C01799=1037.388,344.566,-126.186,172.352,44.021,158.561
C01800=1037.395,344.814,-126.222,172.357,44.023,158.563
C01801=1037.403,345.061,-126.259,172.364,44.026,158.564
C01802=1037.410,345.308,-126.297,172.369,44.028,158.565
C01803=1037.418,345.555,-126.334,172.375,44.031,158.566
C01804=1037.425,345.802,-126.371,172.380,44.033,158.567
C01805=1037.433,346.049,-126.408,172.385,44.036,158.568
C01806=1037.440,346.296,-126.445,172.391,44.039,158.569
C01807=1037.447,346.544,-126.483,172.396,44.041,158.570
C01808=1037.455,346.790,-126.520,172.402,44.043,158.571
C01809=1037.463,347.038,-126.557,172.408,44.046,158.573
C01810=1037.470,347.284,-126.594,172.413,44.049,158.574
C01811=1037.478,347.531,-126.632,172.419,44.051,158.575
C01812=1037.486,347.779,-126.669,172.424,44.054,158.576
C01813=1037.494,348.026,-126.706,172.431,44.057,158.577
C01814=1037.501,348.273,-126.744,172.436,44.059,158.578
C01815=1037.513,348.639,-126.800,172.444,44.063,158.580
C01816=1037.524,349.005,-126.855,172.452,44.067,158.581
C01817=1037.535,349.371,-126.911,172.461,44.071,158.583
C01818=1037.546,349.738,-126.966,172.470,44.075,158.585
C01819=1037.554,349.984,-127.004,172.475,44.077,158.586
C01820=1037.561,350.231,-127.042,172.480,44.080,158.587
C01821=1037.569,350.478,-127.079,172.487,44.083,158.588
C01822=1037.577,350.725,-127.117,172.492,44.085,158.589
C01823=1037.584,350.973,-127.155,172.498,44.089,158.591
C01824=1037.592,351.220,-127.192,172.503,44.092,158.592
C01825=1037.599,351.466,-127.231,172.510,44.094,158.593
C01826=1037.607,351.714,-127.269,172.515,44.097,158.594
C01827=1037.615,351.960,-127.306,172.521,44.100,158.595
C01828=1037.623,352.207,-127.344,172.526,44.102,158.596
C01829=1037.631,352.455,-127.382,172.533,44.105,158.598
C01830=1037.638,352.702,-127.420,172.538,44.108,158.599
C01831=1037.645,352.948,-127.458,172.544,44.111,158.600
C01832=1037.653,353.196,-127.496,172.550,44.114,158.601
C01833=1037.661,353.443,-127.534,172.556,44.116,158.602
C01834=1037.668,353.689,-127.573,172.561,44.119,158.604
C01835=1037.677,353.937,-127.610,172.568,44.122,158.605
C01836=1037.685,354.183,-127.648,172.574,44.125,158.606
C01837=1037.692,354.431,-127.686,172.579,44.128,158.607
C01838=1037.700,354.678,-127.724,172.586,44.130,158.608
C01839=1037.708,354.924,-127.762,172.591,44.134,158.610
C01840=1037.716,355.171,-127.801,172.598,44.136,158.611
C01841=1037.723,355.418,-127.839,172.603,44.139,158.612
C01842=1037.731,355.666,-127.877,172.609,44.142,158.613
C01843=1037.739,355.912,-127.915,172.616,44.145,158.615
C01844=1037.747,356.159,-127.953,172.621,44.148,158.616
C01845=1037.754,356.406,-127.992,172.628,44.151,158.617
C01846=1037.762,356.653,-128.031,172.633,44.154,158.619
C01847=1037.770,356.900,-128.069,172.639,44.157,158.620
C01848=1037.778,357.147,-128.108,172.646,44.160,158.621
C01849=1037.786,357.393,-128.146,172.651,44.163,158.622
C01850=1037.794,357.641,-128.185,172.658,44.166,158.624
C01851=1037.801,357.887,-128.223,172.663,44.168,158.625
C01852=1037.810,358.134,-128.261,172.670,44.172,158.626
C01853=1037.818,358.381,-128.300,172.676,44.175,158.627
C01854=1037.825,358.628,-128.338,172.681,44.178,158.629
C01855=1037.833,358.875,-128.377,172.688,44.181,158.630
C01856=1037.841,359.122,-128.415,172.694,44.184,158.631
C01857=1037.848,359.369,-128.454,172.700,44.187,158.632
C01858=1037.857,359.616,-128.494,172.706,44.190,158.634
C01859=1037.864,359.862,-128.532,172.713,44.193,158.635
C01860=1037.873,360.110,-128.571,172.718,44.196,158.636
C01861=1037.881,360.356,-128.610,172.725,44.199,158.638
C01862=1037.889,360.603,-128.648,172.731,44.202,158.639
C01863=1037.897,360.850,-128.687,172.737,44.205,158.640
C01864=1037.904,361.097,-128.727,172.744,44.208,158.642
C01865=1037.912,361.343,-128.765,172.750,44.212,158.643
C01866=1037.920,361.591,-128.804,172.757,44.215,158.644
C01867=1037.929,361.837,-128.843,172.762,44.218,158.646
C01868=1037.937,362.084,-128.881,172.769,44.221,158.647
C01869=1037.944,362.331,-128.921,172.775,44.225,158.648
C01870=1037.952,362.578,-128.960,172.782,44.228,158.650
C01871=1037.964,362.950,-129.019,172.791,44.233,158.652
C01872=1037.975,363.322,-129.078,172.801,44.237,158.654
C01873=1037.988,363.694,-129.138,172.811,44.242,158.656
C01874=1037.999,364.067,-129.197,172.819,44.248,158.658
C01875=1038.008,364.313,-129.236,172.826,44.251,158.659
C01876=1038.016,364.560,-129.276,172.833,44.254,158.661
C01877=1038.023,364.806,-129.315,172.839,44.258,158.662
C01878=1038.031,365.053,-129.355,172.846,44.261,158.664
C01879=1038.039,365.300,-129.393,172.852,44.264,158.665
C01880=1038.048,365.547,-129.433,172.858,44.267,158.666
C01881=1038.056,365.794,-129.473,172.865,44.271,158.668
C01882=1038.064,366.040,-129.512,172.872,44.274,158.669
C01883=1038.072,366.287,-129.552,172.877,44.277,158.671
C01884=1038.080,366.534,-129.591,172.884,44.281,158.672
C01885=1038.088,366.781,-129.631,172.891,44.284,158.674
C01886=1038.096,367.027,-129.670,172.897,44.288,158.675
C01887=1038.104,367.274,-129.710,172.904,44.291,158.676
C01888=1038.113,367.521,-129.750,172.911,44.295,158.678
C01889=1038.121,367.767,-129.789,172.917,44.298,158.679
C01890=1038.129,368.014,-129.829,172.924,44.302,158.681
C01891=1038.137,368.260,-129.869,172.931,44.305,158.682
C01892=1038.145,368.507,-129.909,172.938,44.308,158.684
C01893=1038.154,368.754,-129.948,172.943,44.312,158.685
C01894=1038.161,369.001,-129.988,172.950,44.315,158.687
C01895=1038.170,369.247,-130.027,172.957,44.318,158.688
C01896=1038.178,369.493,-130.068,172.964,44.322,158.690
C01897=1038.186,369.740,-130.107,172.971,44.326,158.691
C01898=1038.195,369.988,-130.148,172.977,44.329,158.692
C01899=1038.203,370.234,-130.188,172.984,44.333,158.694
C01900=1038.211,370.480,-130.228,172.991,44.336,158.696
C01901=1038.219,370.727,-130.268,172.998,44.340,158.697
C01902=1038.228,370.973,-130.308,173.005,44.343,158.699
C01903=1038.236,371.220,-130.348,173.011,44.347,158.700
C01904=1038.243,371.467,-130.388,173.018,44.351,158.702
C01905=1038.251,371.713,-130.429,173.025,44.355,158.703
C01906=1038.260,371.960,-130.470,173.032,44.358,158.705
C01907=1038.268,372.206,-130.509,173.039,44.362,158.706
C01908=1038.276,372.453,-130.550,173.046,44.366,158.708
C01909=1038.285,372.699,-130.590,173.053,44.369,158.709
C01910=1038.293,372.947,-130.631,173.059,44.373,158.711
C01911=1038.302,373.193,-130.671,173.066,44.377,158.712
C01912=1038.310,373.439,-130.711,173.073,44.380,158.714
C01913=1038.318,373.685,-130.752,173.080,44.384,158.716
C01914=1038.326,373.932,-130.793,173.087,44.388,158.717
C01915=1038.334,374.179,-130.833,173.094,44.391,158.719
C01916=1038.343,374.425,-130.873,173.101,44.395,158.720
C01917=1038.351,374.672,-130.914,173.108,44.399,158.722
C01918=1038.359,374.918,-130.955,173.115,44.403,158.724
C01919=1038.367,375.165,-130.995,173.122,44.406,158.725
C01920=1038.376,375.412,-131.036,173.130,44.411,158.727
C01921=1038.384,375.658,-131.077,173.137,44.414,158.728
C01922=1038.393,375.904,-131.117,173.144,44.418,158.730
C01923=1038.401,376.151,-131.158,173.151,44.422,158.732
C01924=1038.410,376.397,-131.199,173.158,44.426,158.733
C01925=1038.418,376.643,-131.240,173.165,44.429,158.735
C01926=1038.426,376.890,-131.281,173.172,44.433,158.736
C01927=1038.441,377.283,-131.346,173.184,44.439,158.739
C01928=1038.454,377.675,-131.410,173.195,44.446,158.742
C01929=1038.468,378.068,-131.476,173.207,44.452,158.744
C01930=1038.482,378.461,-131.541,173.218,44.458,158.747
C01931=1038.489,378.707,-131.583,173.225,44.462,158.749
C01932=1038.498,378.954,-131.624,173.233,44.467,158.750
C01933=1038.506,379.200,-131.665,173.240,44.470,158.752
C01934=1038.515,379.447,-131.706,173.247,44.474,158.754
C01935=1038.523,379.692,-131.748,173.254,44.478,158.755
C01936=1038.532,379.939,-131.789,173.261,44.483,158.757
C01937=1038.541,380.184,-131.831,173.270,44.487,158.759
C01938=1038.549,380.431,-131.872,173.277,44.491,158.761
C01939=1038.558,380.677,-131.913,173.284,44.495,158.762
C01940=1038.566,380.923,-131.955,173.292,44.499,158.764
C01941=1038.574,381.169,-131.997,173.299,44.503,158.766
C01942=1038.583,381.416,-132.038,173.306,44.507,158.768
C01943=1038.591,381.662,-132.079,173.315,44.511,158.769
C01944=1038.600,381.908,-132.121,173.322,44.516,158.771
C01945=1038.609,382.155,-132.162,173.329,44.520,158.773
C01946=1038.618,382.401,-132.204,173.336,44.524,158.775
C01947=1038.625,382.647,-132.246,173.344,44.528,158.776
C01948=1038.634,382.893,-132.288,173.352,44.532,158.778
C01949=1038.643,383.140,-132.330,173.360,44.537,158.780
C01950=1038.652,383.386,-132.371,173.367,44.541,158.782
C01951=1038.661,383.633,-132.413,173.374,44.545,158.783
C01952=1038.669,383.878,-132.454,173.383,44.549,158.785
C01953=1038.678,384.125,-132.497,173.390,44.554,158.787
C01954=1038.687,384.371,-132.538,173.397,44.558,158.789
C01955=1038.696,384.618,-132.580,173.406,44.562,158.791
C01956=1038.704,384.864,-132.622,173.413,44.567,158.793
C01957=1038.714,385.110,-132.664,173.421,44.571,158.794
C01958=1038.722,385.356,-132.707,173.428,44.575,158.796
C01959=1038.731,385.603,-132.748,173.436,44.579,158.798
C01960=1038.740,385.849,-132.790,173.444,44.584,158.800
C01961=1038.749,386.095,-132.832,173.452,44.588,158.802
C01962=1038.758,386.341,-132.874,173.460,44.593,158.804
C01963=1038.766,386.588,-132.916,173.467,44.597,158.805
C01964=1038.775,386.834,-132.959,173.476,44.601,158.807
C01965=1038.784,387.080,-133.001,173.483,44.606,158.809
C01966=1038.794,387.326,-133.043,173.492,44.610,158.811
C01967=1038.802,387.572,-133.085,173.499,44.615,158.813
C01968=1038.811,387.818,-133.128,173.508,44.619,158.815
C01969=1038.820,388.065,-133.169,173.515,44.624,158.817
C01970=1038.829,388.311,-133.213,173.523,44.628,158.819
C01971=1038.838,388.557,-133.255,173.531,44.632,158.821
C01972=1038.847,388.803,-133.297,173.539,44.637,158.823
C01973=1038.856,389.050,-133.340,173.548,44.642,158.825
C01974=1038.865,389.295,-133.382,173.555,44.646,158.826
C01975=1038.873,389.541,-133.426,173.564,44.651,158.828
C01976=1038.883,389.787,-133.468,173.571,44.655,158.830
C01977=1038.892,390.034,-133.511,173.580,44.660,158.832
C01978=1038.901,390.280,-133.553,173.588,44.665,158.834
C01979=1038.909,390.526,-133.596,173.596,44.670,158.836
C01980=1038.918,390.772,-133.639,173.604,44.674,158.838
C01981=1038.928,391.019,-133.682,173.613,44.679,158.840
C01982=1038.937,391.264,-133.724,173.621,44.684,158.842
C01983=1038.945,391.477,-133.762,173.627,44.687,158.844
C01984=1038.952,391.691,-133.799,173.635,44.692,158.846
C01985=1038.959,391.904,-133.837,173.642,44.696,158.847
C01986=1038.967,392.117,-133.874,173.649,44.700,158.849
C01987=1038.976,392.331,-133.912,173.657,44.704,158.851
C01988=1038.983,392.544,-133.949,173.664,44.709,158.853
C01989=1038.991,392.757,-133.986,173.672,44.713,158.855
C01990=1038.999,392.971,-134.024,173.679,44.717,158.856
C01991=1039.009,393.217,-134.067,173.687,44.721,158.858
C01992=1039.017,393.463,-134.110,173.696,44.726,158.861
C01993=1039.026,393.709,-134.154,173.704,44.731,158.863
C01994=1039.036,393.955,-134.196,173.712,44.736,158.865
C01995=1039.045,394.201,-134.240,173.721,44.741,158.867
C01996=1039.054,394.447,-134.283,173.730,44.746,158.869
C01997=1039.064,394.693,-134.327,173.737,44.751,158.871
C01998=1039.072,394.939,-134.370,173.746,44.756,158.873
C01999=1039.082,395.185,-134.414,173.755,44.761,158.875
C02000=1039.091,395.430,-134.457,173.764,44.766,158.877
C02001=1039.100,395.677,-134.501,173.772,44.771,158.879
C02002=1039.109,395.922,-134.544,173.781,44.776,158.882
C02003=1039.119,396.168,-134.588,173.790,44.781,158.884
C02004=1039.127,396.414,-134.632,173.799,44.786,158.886
C02005=1039.136,396.660,-134.676,173.807,44.791,158.888
C02006=1039.147,396.906,-134.719,173.815,44.796,158.890
C02007=1039.155,397.152,-134.763,173.824,44.801,158.892
C02008=1039.165,397.398,-134.807,173.833,44.806,158.895
C02009=1039.174,397.644,-134.851,173.842,44.811,158.897
C02010=1039.183,397.889,-134.895,173.851,44.816,158.899
C02011=1039.192,398.136,-134.939,173.860,44.821,158.901
C02012=1039.203,398.381,-134.982,173.869,44.826,158.903
C02013=1039.212,398.627,-135.027,173.878,44.832,158.906
C02014=1039.221,398.873,-135.070,173.887,44.837,158.908
C02015=1039.231,399.118,-135.115,173.896,44.842,158.910
C02016=1039.240,399.365,-135.159,173.904,44.848,158.912
C02017=1039.249,399.611,-135.203,173.913,44.853,158.914
C02018=1039.259,399.857,-135.247,173.922,44.858,158.917
C02019=1039.268,400.102,-135.292,173.931,44.863,158.919
C02020=1039.277,400.348,-135.336,173.940,44.868,158.921
C02021=1039.287,400.594,-135.380,173.949,44.874,158.924
C02022=1039.296,400.839,-135.425,173.958,44.879,158.926
C02023=1039.306,401.086,-135.469,173.968,44.884,158.928
C02024=1039.316,401.331,-135.514,173.978,44.890,158.931
C02025=1039.325,401.577,-135.558,173.987,44.895,158.933
C02026=1039.335,401.823,-135.603,173.996,44.901,158.935
C02027=1039.344,402.068,-135.648,174.005,44.906,158.938
C02028=1039.354,402.314,-135.692,174.014,44.911,158.940
C02029=1039.363,402.560,-135.737,174.023,44.917,158.942
C02030=1039.373,402.805,-135.781,174.032,44.922,158.945
C02031=1039.382,403.051,-135.827,174.042,44.928,158.947
C02032=1039.392,403.298,-135.871,174.051,44.934,158.949
C02033=1039.402,403.544,-135.916,174.061,44.939,158.952
C02034=1039.412,403.789,-135.961,174.070,44.944,158.954
C02035=1039.421,404.035,-136.006,174.080,44.950,158.957
C02036=1039.430,404.280,-136.051,174.089,44.956,158.959
C02037=1039.440,404.526,-136.096,174.098,44.961,158.961
C02038=1039.450,404.771,-136.141,174.108,44.967,158.964
C02039=1039.459,405.018,-136.187,174.118,44.973,158.966
C02040=1039.469,405.263,-136.232,174.127,44.978,158.969
C02041=1039.479,405.508,-136.277,174.137,44.984,158.971
C02042=1039.488,405.754,-136.322,174.147,44.989,158.974
C02043=1039.498,405.978,-136.363,174.155,44.995,158.976
C02044=1039.506,406.201,-136.405,174.164,45.000,158.978
C02045=1039.515,406.424,-136.446,174.173,45.005,158.981
C02046=1039.525,406.647,-136.487,174.182,45.010,158.983
C02047=1039.533,406.870,-136.529,174.190,45.016,158.985
C02048=1039.542,407.093,-136.569,174.199,45.021,158.987
C02049=1039.551,407.317,-136.611,174.208,45.026,158.990
C02050=1039.560,407.540,-136.653,174.218,45.032,158.992
C02051=1039.570,407.786,-136.698,174.227,45.038,158.995
C02052=1039.580,408.031,-136.744,174.238,45.043,158.997
C02053=1039.590,408.277,-136.789,174.247,45.049,159.000
C02054=1039.599,408.523,-136.835,174.257,45.055,159.002
C02055=1039.609,408.769,-136.880,174.267,45.061,159.005
C02056=1039.620,409.014,-136.926,174.277,45.067,159.007
C02057=1039.629,409.260,-136.972,174.287,45.073,159.010
C02058=1039.640,409.505,-137.018,174.297,45.079,159.013
C02059=1039.650,409.750,-137.064,174.307,45.084,159.015
C02060=1039.660,409.997,-137.110,174.318,45.090,159.018
C02061=1039.670,410.242,-137.156,174.327,45.097,159.020
C02062=1039.680,410.487,-137.201,174.338,45.102,159.023
C02063=1039.690,410.733,-137.248,174.348,45.109,159.026
C02064=1039.701,410.979,-137.294,174.358,45.115,159.028
C02065=1039.711,411.223,-137.339,174.369,45.120,159.031
C02066=1039.721,411.469,-137.386,174.379,45.127,159.034
C02067=1039.731,411.715,-137.431,174.389,45.133,159.037
C02068=1039.741,411.960,-137.479,174.400,45.139,159.039
C02069=1039.751,412.206,-137.525,174.410,45.145,159.042
C02070=1039.762,412.452,-137.571,174.420,45.152,159.045
C02071=1039.772,412.696,-137.618,174.431,45.158,159.047
C02072=1039.781,412.942,-137.664,174.441,45.164,159.050
C02073=1039.792,413.188,-137.710,174.452,45.170,159.053
C02074=1039.802,413.433,-137.758,174.462,45.176,159.056
C02075=1039.812,413.679,-137.804,174.473,45.183,159.058
C02076=1039.823,413.924,-137.851,174.484,45.189,159.061
C02077=1039.833,414.169,-137.898,174.494,45.196,159.064
C02078=1039.843,414.415,-137.944,174.505,45.202,159.067
C02079=1039.854,414.660,-137.991,174.516,45.208,159.070
C02080=1039.864,414.905,-138.038,174.527,45.215,159.073
C02081=1039.874,415.151,-138.085,174.538,45.221,159.075
C02082=1039.884,415.397,-138.132,174.548,45.228,159.078
C02083=1039.895,415.642,-138.179,174.559,45.234,159.081
C02084=1039.905,415.887,-138.226,174.570,45.241,159.084
C02085=1039.916,416.132,-138.273,174.581,45.247,159.087
C02086=1039.927,416.378,-138.320,174.592,45.254,159.090
C02087=1039.937,416.623,-138.367,174.603,45.260,159.093
C02088=1039.948,416.868,-138.414,174.614,45.266,159.096
C02089=1039.959,417.113,-138.461,174.625,45.273,159.099
C02090=1039.969,417.359,-138.508,174.636,45.280,159.102
C02091=1039.980,417.605,-138.556,174.647,45.286,159.104
C02092=1039.990,417.850,-138.603,174.658,45.293,159.107
C02093=1040.001,418.095,-138.651,174.670,45.300,159.110
C02094=1040.011,418.341,-138.699,174.681,45.306,159.113
C02095=1040.021,418.585,-138.747,174.692,45.313,159.116
C02096=1040.032,418.831,-138.794,174.704,45.320,159.119
C02097=1040.043,419.076,-138.842,174.715,45.327,159.123
C02098=1040.053,419.321,-138.889,174.726,45.334,159.126
C02099=1040.064,419.566,-138.938,174.738,45.340,159.129
C02100=1040.075,419.811,-138.984,174.749,45.347,159.132
C02101=1040.086,420.057,-139.032,174.761,45.354,159.135
C02102=1040.097,420.301,-139.080,174.772,45.361,159.138
C02103=1040.106,420.529,-139.125,174.783,45.367,159.141
C02104=1040.116,420.756,-139.169,174.793,45.374,159.144
C02105=1040.126,420.985,-139.214,174.804,45.380,159.146
C02106=1040.136,421.211,-139.259,174.815,45.387,159.149
C02107=1040.146,421.439,-139.303,174.826,45.393,159.152
C02108=1040.156,421.666,-139.348,174.837,45.399,159.155
C02109=1040.167,421.894,-139.393,174.848,45.406,159.158
C02110=1040.176,422.121,-139.437,174.859,45.412,159.161
C02111=1040.187,422.367,-139.486,174.871,45.419,159.164
C02112=1040.198,422.611,-139.534,174.883,45.426,159.168
C02113=1040.209,422.856,-139.583,174.895,45.434,159.171
C02114=1040.220,423.101,-139.631,174.907,45.440,159.174
C02115=1040.232,423.347,-139.679,174.919,45.448,159.177
C02116=1040.243,423.592,-139.728,174.931,45.455,159.181
C02117=1040.253,423.836,-139.776,174.943,45.462,159.184
C02118=1040.265,424.082,-139.824,174.955,45.469,159.187
C02119=1040.276,424.326,-139.873,174.968,45.476,159.190
C02120=1040.287,424.572,-139.922,174.979,45.484,159.194
C02121=1040.298,424.816,-139.971,174.992,45.491,159.197
C02122=1040.309,425.061,-140.020,175.005,45.498,159.200
C02123=1040.320,425.307,-140.069,175.016,45.506,159.204
C02124=1040.332,425.552,-140.118,175.029,45.513,159.207
C02125=1040.343,425.796,-140.167,175.042,45.520,159.211
C02126=1040.354,426.041,-140.216,175.054,45.528,159.214
C02127=1040.365,426.286,-140.265,175.066,45.535,159.217
C02128=1040.377,426.531,-140.314,175.079,45.543,159.221
C02129=1040.388,426.776,-140.363,175.092,45.550,159.224
C02130=1040.399,427.021,-140.413,175.104,45.557,159.228
C02131=1040.410,427.265,-140.462,175.117,45.565,159.231
C02132=1040.421,427.510,-140.511,175.130,45.572,159.234
C02133=1040.433,427.756,-140.560,175.143,45.580,159.238
C02134=1040.444,428.001,-140.610,175.156,45.588,159.242
C02135=1040.456,428.245,-140.660,175.168,45.595,159.245
C02136=1040.467,428.490,-140.709,175.182,45.603,159.249
C02137=1040.478,428.735,-140.759,175.194,45.610,159.252
C02138=1040.490,428.979,-140.808,175.207,45.618,159.256
C02139=1040.501,429.224,-140.858,175.220,45.626,159.259
C02140=1040.513,429.469,-140.908,175.233,45.634,159.263
C02141=1040.524,429.714,-140.958,175.246,45.642,159.267
C02142=1040.536,429.958,-141.007,175.260,45.649,159.270
C02143=1040.547,430.204,-141.058,175.273,45.657,159.274
C02144=1040.559,430.448,-141.108,175.286,45.665,159.278
C02145=1040.570,430.692,-141.158,175.300,45.673,159.281
C02146=1040.582,430.937,-141.208,175.313,45.681,159.285
C02147=1040.593,431.181,-141.259,175.326,45.689,159.289
C02148=1040.605,431.426,-141.309,175.339,45.697,159.292
C02149=1040.617,431.671,-141.359,175.353,45.704,159.296
C02150=1040.629,431.915,-141.409,175.367,45.713,159.300
C02151=1040.640,432.161,-141.460,175.380,45.720,159.303
C02152=1040.652,432.405,-141.510,175.394,45.728,159.307
C02153=1040.664,432.649,-141.561,175.407,45.736,159.311
C02154=1040.676,432.894,-141.611,175.422,45.745,159.315
C02155=1040.688,433.139,-141.662,175.435,45.752,159.319
C02156=1040.700,433.383,-141.712,175.449,45.761,159.322
C02157=1040.711,433.628,-141.763,175.463,45.769,159.326
C02158=1040.724,433.872,-141.814,175.477,45.777,159.330
C02159=1040.736,434.117,-141.864,175.491,45.785,159.334
C02160=1040.748,434.361,-141.915,175.505,45.794,159.338
C02161=1040.760,434.606,-141.966,175.520,45.802,159.342
C02162=1040.772,434.850,-142.016,175.533,45.810,159.346
C02163=1040.783,435.085,-142.065,175.547,45.817,159.350
C02164=1040.795,435.319,-142.115,175.561,45.826,159.353
C02165=1040.807,435.554,-142.164,175.574,45.834,159.357
C02166=1040.818,435.788,-142.213,175.588,45.842,159.361
C02167=1040.829,436.022,-142.262,175.602,45.850,159.365
C02168=1040.842,436.256,-142.311,175.616,45.858,159.369
C02169=1040.853,436.491,-142.361,175.630,45.866,159.373
C02170=1040.865,436.726,-142.409,175.644,45.874,159.377
C02171=1040.877,436.969,-142.462,175.659,45.882,159.381
C02172=1040.889,437.214,-142.513,175.674,45.891,159.385
C02173=1040.901,437.458,-142.564,175.688,45.899,159.389
C02174=1040.914,437.702,-142.616,175.703,45.908,159.393
C02175=1040.926,437.947,-142.668,175.718,45.917,159.397
C02176=1040.939,438.191,-142.720,175.733,45.925,159.401
C02177=1040.951,438.436,-142.771,175.748,45.934,159.406
C02178=1040.963,438.680,-142.823,175.763,45.943,159.410
C02179=1040.976,438.924,-142.876,175.777,45.951,159.414
C02180=1040.988,439.168,-142.927,175.793,45.960,159.418
C02181=1041.001,439.412,-142.980,175.808,45.969,159.423
C02182=1041.013,439.657,-143.031,175.823,45.978,159.427
C02183=1041.026,439.901,-143.084,175.839,45.987,159.431
C02184=1041.038,440.145,-143.136,175.854,45.996,159.435
C02185=1041.051,440.390,-143.188,175.869,46.005,159.440
C02186=1041.063,440.633,-143.241,175.885,46.013,159.444
C02187=1041.076,440.878,-143.294,175.900,46.022,159.448
C02188=1041.088,441.122,-143.346,175.916,46.031,159.453
C02189=1041.101,441.366,-143.398,175.931,46.040,159.457
C02190=1041.114,441.610,-143.451,175.948,46.049,159.462
C02191=1041.126,441.854,-143.504,175.963,46.058,159.466
C02192=1041.140,442.098,-143.557,175.979,46.067,159.470
C02193=1041.153,442.342,-143.609,175.995,46.076,159.475
C02194=1041.166,442.586,-143.662,176.011,46.086,159.480
C02195=1041.179,442.830,-143.715,176.026,46.095,159.484
C02196=1041.191,443.074,-143.767,176.043,46.104,159.489
C02197=1041.205,443.318,-143.820,176.059,46.113,159.493
C02198=1041.218,443.562,-143.874,176.076,46.122,159.498
C02199=1041.231,443.806,-143.927,176.091,46.131,159.502
C02200=1041.244,444.050,-143.980,176.108,46.141,159.507
C02201=1041.257,444.294,-144.033,176.124,46.150,159.512
C02202=1041.270,444.538,-144.086,176.141,46.159,159.516
C02203=1041.283,444.781,-144.140,176.157,46.169,159.521
C02204=1041.296,445.023,-144.193,176.174,46.178,159.526
C02205=1041.311,445.266,-144.245,176.191,46.187,159.530
C02206=1041.326,445.511,-144.297,176.207,46.196,159.535
C02207=1041.341,445.754,-144.348,176.224,46.206,159.540
C02208=1041.356,445.997,-144.399,176.241,46.214,159.544
C02209=1041.374,446.241,-144.450,176.258,46.223,159.549
C02210=1041.390,446.485,-144.500,176.275,46.232,159.553
C02211=1041.408,446.729,-144.549,176.292,46.240,159.558
C02212=1041.427,446.973,-144.599,176.309,46.248,159.562
C02213=1041.446,447.217,-144.647,176.327,46.257,159.567
C02214=1041.465,447.462,-144.695,176.344,46.265,159.571
C02215=1041.485,447.706,-144.743,176.361,46.273,159.576
C02216=1041.506,447.950,-144.790,176.380,46.281,159.580
C02217=1041.527,448.195,-144.837,176.397,46.289,159.585
C02218=1041.549,448.440,-144.884,176.415,46.296,159.589
C02219=1041.571,448.684,-144.930,176.432,46.305,159.594
C02220=1041.595,448.929,-144.975,176.450,46.312,159.598
C02221=1041.619,449.175,-145.019,176.468,46.320,159.602
C02222=1041.643,449.419,-145.064,176.486,46.327,159.607
C02223=1041.671,449.706,-145.115,176.507,46.335,159.612
C02224=1041.702,449.993,-145.166,176.529,46.344,159.617
C02225=1041.732,450.280,-145.216,176.550,46.352,159.622
C02226=1041.764,450.567,-145.265,176.571,46.360,159.627
C02227=1041.791,450.813,-145.307,176.590,46.367,159.631
C02228=1041.820,451.059,-145.348,176.608,46.373,159.635
C02229=1041.849,451.304,-145.389,176.627,46.380,159.639
C02230=1041.878,451.549,-145.429,176.645,46.387,159.644
C02231=1041.579,451.594,-145.745,176.648,46.464,159.667
C02232=1041.550,451.349,-145.705,176.629,46.458,159.663
C02233=1041.521,451.104,-145.664,176.611,46.452,159.659
C02234=1041.493,450.858,-145.623,176.592,46.445,159.655
C02235=1041.465,450.612,-145.581,176.573,46.438,159.650
C02236=1041.435,450.341,-145.535,176.553,46.431,159.646
C02237=1041.405,450.068,-145.488,176.533,46.423,159.641
C02238=1041.376,449.797,-145.440,176.513,46.415,159.636
C02239=1041.349,449.525,-145.392,176.492,46.407,159.631
C02240=1041.324,449.280,-145.348,176.474,46.400,159.627
C02241=1041.300,449.035,-145.302,176.456,46.392,159.623
C02242=1041.276,448.790,-145.258,176.438,46.385,159.618
C02243=1041.254,448.546,-145.213,176.420,46.378,159.614
C02244=1041.231,448.301,-145.166,176.403,46.370,159.609
C02245=1041.210,448.056,-145.120,176.385,46.362,159.605
C02246=1041.189,447.812,-145.072,176.368,46.354,159.601
C02247=1041.169,447.568,-145.025,176.349,46.346,159.596
C02248=1041.148,447.323,-144.977,176.332,46.338,159.592
C02249=1041.130,447.079,-144.929,176.315,46.330,159.587
C02250=1041.111,446.834,-144.880,176.298,46.322,159.583
C02251=1041.093,446.591,-144.831,176.280,46.313,159.578
C02252=1041.075,446.346,-144.781,176.263,46.305,159.574
C02253=1041.058,446.103,-144.731,176.246,46.296,159.569
C02254=1041.041,445.859,-144.680,176.229,46.288,159.564
C02255=1041.026,445.616,-144.629,176.213,46.279,159.560
C02256=1041.011,445.372,-144.577,176.195,46.270,159.555
C02257=1040.996,445.128,-144.525,176.178,46.261,159.551
C02258=1040.983,444.886,-144.473,176.162,46.252,159.546
C02259=1040.969,444.642,-144.420,176.145,46.243,159.541
C02260=1040.956,444.399,-144.366,176.129,46.233,159.537
C02261=1040.942,444.155,-144.313,176.112,46.224,159.532
C02262=1040.929,443.911,-144.260,176.095,46.215,159.527
C02263=1040.916,443.667,-144.207,176.079,46.206,159.523
C02264=1040.903,443.423,-144.154,176.063,46.196,159.518
C02265=1040.891,443.179,-144.101,176.047,46.187,159.514
C02266=1040.878,442.935,-144.047,176.031,46.178,159.509
C02267=1040.864,442.691,-143.994,176.014,46.169,159.504
C02268=1040.852,442.447,-143.942,175.999,46.160,159.500
C02269=1040.839,442.203,-143.889,175.982,46.151,159.495
C02270=1040.826,441.960,-143.836,175.966,46.142,159.491
C02271=1040.813,441.715,-143.783,175.951,46.133,159.486
C02272=1040.800,441.471,-143.730,175.935,46.124,159.482
C02273=1040.787,441.226,-143.678,175.919,46.115,159.478
C02274=1040.774,440.983,-143.626,175.903,46.107,159.473
C02275=1040.761,440.739,-143.573,175.888,46.098,159.469
C02276=1040.749,440.495,-143.521,175.872,46.089,159.464
C02277=1040.736,440.250,-143.468,175.857,46.080,159.460
C02278=1040.724,440.006,-143.416,175.842,46.071,159.456
C02279=1040.711,439.762,-143.364,175.825,46.062,159.451
C02280=1040.699,439.517,-143.311,175.811,46.054,159.447
C02281=1040.686,439.273,-143.259,175.795,46.045,159.443
C02282=1040.674,439.030,-143.208,175.780,46.036,159.439
C02283=1040.661,438.785,-143.155,175.764,46.027,159.434
C02284=1040.649,438.541,-143.104,175.750,46.019,159.430
C02285=1040.637,438.297,-143.051,175.735,46.010,159.426
C02286=1040.624,438.052,-142.999,175.720,46.002,159.422
C02287=1040.612,437.808,-142.948,175.705,45.993,159.418
C02288=1040.599,437.564,-142.896,175.690,45.985,159.414
C02289=1040.587,437.320,-142.845,175.675,45.976,159.409
C02290=1040.575,437.074,-142.793,175.661,45.968,159.405
C02291=1040.563,436.831,-142.741,175.646,45.959,159.401
C02292=1040.551,436.596,-142.692,175.631,45.951,159.397
C02293=1040.538,436.361,-142.642,175.618,45.943,159.393
C02294=1040.527,436.126,-142.593,175.603,45.935,159.389
C02295=1040.515,435.891,-142.543,175.590,45.927,159.386
C02296=1040.504,435.656,-142.494,175.575,45.919,159.382
C02297=1040.492,435.420,-142.445,175.562,45.911,159.378
C02298=1040.480,435.185,-142.395,175.548,45.903,159.374
C02299=1040.469,434.950,-142.347,175.534,45.895,159.370
C02300=1040.456,434.706,-142.296,175.520,45.887,159.366
C02301=1040.445,434.461,-142.245,175.505,45.879,159.362
C02302=1040.432,434.217,-142.194,175.492,45.870,159.358
C02303=1040.420,433.972,-142.143,175.478,45.863,159.355
C02304=1040.408,433.728,-142.093,175.463,45.855,159.351
C02305=1040.397,433.484,-142.042,175.450,45.846,159.347
C02306=1040.384,433.239,-141.992,175.435,45.838,159.343
C02307=1040.372,432.994,-141.940,175.422,45.830,159.339
C02308=1040.360,432.749,-141.890,175.407,45.822,159.335
C02309=1040.349,432.505,-141.840,175.394,45.815,159.332
C02310=1040.337,432.260,-141.790,175.380,45.806,159.328
C02311=1040.325,432.016,-141.738,175.367,45.799,159.324
C02312=1040.313,431.772,-141.689,175.353,45.791,159.320
C02313=1040.302,431.526,-141.638,175.339,45.783,159.317
C02314=1040.290,431.282,-141.588,175.326,45.775,159.313
C02315=1040.278,431.037,-141.537,175.312,45.767,159.309
C02316=1040.266,430.792,-141.487,175.299,45.759,159.305
C02317=1040.255,430.548,-141.437,175.285,45.751,159.302
C02318=1040.243,430.304,-141.387,175.272,45.743,159.298
C02319=1040.232,430.058,-141.337,175.258,45.736,159.294
C02320=1040.220,429.814,-141.288,175.245,45.728,159.291
C02321=1040.209,429.569,-141.237,175.232,45.721,159.287
C02322=1040.197,429.325,-141.187,175.219,45.713,159.283
C02323=1040.186,429.080,-141.138,175.206,45.705,159.280
C02324=1040.174,428.835,-141.087,175.193,45.697,159.276
C02325=1040.163,428.590,-141.038,175.180,45.690,159.273
C02326=1040.152,428.346,-140.988,175.167,45.683,159.269
C02327=1040.141,428.101,-140.938,175.153,45.675,159.266
C02328=1040.129,427.855,-140.889,175.141,45.667,159.262
C02329=1040.117,427.611,-140.839,175.128,45.660,159.259
C02330=1040.106,427.366,-140.790,175.115,45.653,159.255
C02331=1040.095,427.121,-140.741,175.103,45.645,159.252
C02332=1040.084,426.877,-140.692,175.090,45.638,159.248
C02333=1040.072,426.631,-140.642,175.077,45.630,159.245
C02334=1040.060,426.386,-140.593,175.065,45.623,159.241
C02335=1040.049,426.142,-140.544,175.052,45.615,159.238
C02336=1040.038,425.897,-140.495,175.039,45.608,159.235
C02337=1040.027,425.652,-140.446,175.027,45.601,159.231
C02338=1040.016,425.407,-140.397,175.015,45.593,159.228
C02339=1040.004,425.162,-140.348,175.002,45.586,159.225
C02340=1039.994,424.917,-140.299,174.989,45.579,159.221
C02341=1039.982,424.672,-140.250,174.977,45.572,159.218
C02342=1039.971,424.427,-140.201,174.965,45.564,159.214
C02343=1039.960,424.182,-140.153,174.953,45.557,159.211
C02344=1039.949,423.937,-140.105,174.940,45.550,159.208
C02345=1039.938,423.692,-140.056,174.929,45.543,159.205
C02346=1039.927,423.447,-140.007,174.916,45.536,159.201
C02347=1039.916,423.201,-139.958,174.905,45.529,159.198
C02348=1039.904,422.957,-139.910,174.892,45.522,159.195
C02349=1039.893,422.712,-139.862,174.880,45.515,159.192
C02350=1039.883,422.467,-139.814,174.868,45.508,159.188
C02351=1039.872,422.222,-139.765,174.856,45.501,159.185
C02352=1039.862,421.993,-139.720,174.845,45.494,159.182
C02353=1039.851,421.764,-139.675,174.834,45.488,159.179
C02354=1039.841,421.536,-139.630,174.822,45.482,159.176
C02355=1039.831,421.307,-139.585,174.812,45.475,159.173
C02356=1039.821,421.079,-139.540,174.801,45.469,159.170
C02357=1039.811,420.850,-139.496,174.790,45.462,159.167
C02358=1039.801,420.622,-139.451,174.779,45.456,159.165
C02359=1039.791,420.394,-139.406,174.768,45.450,159.162
C02360=1039.780,420.148,-139.358,174.757,45.443,159.159
C02361=1039.770,419.903,-139.311,174.745,45.436,159.155
C02362=1039.758,419.658,-139.262,174.734,45.429,159.152
C02363=1039.748,419.413,-139.214,174.722,45.422,159.149
C02364=1039.737,419.167,-139.167,174.711,45.415,159.146
C02365=1039.727,418.923,-139.119,174.699,45.409,159.143
C02366=1039.716,418.677,-139.072,174.688,45.402,159.140
C02367=1039.705,418.432,-139.023,174.677,45.396,159.137
C02368=1039.695,418.187,-138.976,174.665,45.389,159.134
C02369=1039.685,417.942,-138.928,174.654,45.382,159.131
C02370=1039.674,417.696,-138.881,174.642,45.376,159.128
C02371=1039.663,417.451,-138.834,174.631,45.369,159.125
C02372=1039.653,417.206,-138.787,174.620,45.363,159.122
C02373=1039.642,416.960,-138.739,174.609,45.356,159.119
C02374=1039.632,416.714,-138.692,174.598,45.350,159.116
C02375=1039.621,416.469,-138.645,174.587,45.343,159.113
C02376=1039.611,416.224,-138.598,174.576,45.337,159.111
C02377=1039.600,415.978,-138.551,174.565,45.330,159.108
C02378=1039.589,415.733,-138.504,174.554,45.324,159.105
C02379=1039.579,415.488,-138.457,174.543,45.318,159.102
C02380=1039.569,415.243,-138.410,174.532,45.311,159.099
C02381=1039.558,414.998,-138.363,174.521,45.305,159.096
C02382=1039.547,414.752,-138.316,174.510,45.299,159.093
C02383=1039.538,414.506,-138.269,174.500,45.292,159.091
C02384=1039.527,414.261,-138.223,174.489,45.286,159.088
C02385=1039.516,414.016,-138.175,174.478,45.279,159.085
C02386=1039.507,413.770,-138.129,174.468,45.273,159.082
C02387=1039.496,413.525,-138.082,174.457,45.267,159.079
C02388=1039.486,413.279,-138.036,174.446,45.261,159.077
C02389=1039.476,413.034,-137.989,174.436,45.255,159.074
C02390=1039.465,412.789,-137.943,174.425,45.248,159.071
C02391=1039.455,412.543,-137.895,174.415,45.242,159.068
C02392=1039.445,412.298,-137.849,174.404,45.236,159.065
C02393=1039.435,412.052,-137.803,174.394,45.230,159.063
C02394=1039.425,411.807,-137.756,174.383,45.224,159.060
C02395=1039.415,411.561,-137.710,174.373,45.217,159.057
C02396=1039.404,411.316,-137.664,174.362,45.212,159.055
C02397=1039.394,411.071,-137.618,174.352,45.206,159.052
C02398=1039.384,410.825,-137.572,174.342,45.199,159.049
C02399=1039.374,410.579,-137.526,174.331,45.194,159.047
C02400=1039.363,410.334,-137.480,174.321,45.188,159.044
C02401=1039.354,410.088,-137.434,174.311,45.181,159.041
C02402=1039.343,409.843,-137.388,174.301,45.176,159.039
C02403=1039.333,409.597,-137.341,174.291,45.170,159.036
C02404=1039.323,409.351,-137.297,174.281,45.164,159.033
C02405=1039.313,409.106,-137.251,174.271,45.158,159.031
C02406=1039.303,408.860,-137.204,174.260,45.152,159.028
C02407=1039.293,408.615,-137.159,174.250,45.147,159.026
C02408=1039.283,408.369,-137.113,174.240,45.141,159.023
C02409=1039.273,408.124,-137.067,174.230,45.135,159.021
C02410=1039.263,407.878,-137.021,174.220,45.129,159.018
C02411=1039.253,407.633,-136.977,174.211,45.123,159.015
C02412=1039.244,407.408,-136.934,174.202,45.117,159.013
C02413=1039.235,407.184,-136.893,174.193,45.113,159.011
C02414=1039.226,406.959,-136.852,174.183,45.107,159.008
C02415=1039.217,406.735,-136.810,174.174,45.102,159.006
C02416=1039.208,406.511,-136.768,174.165,45.097,159.004
C02417=1039.199,406.286,-136.728,174.156,45.092,159.002
C02418=1039.190,406.062,-136.686,174.148,45.086,158.999
C02419=1039.181,405.838,-136.644,174.139,45.082,158.997
C02420=1039.171,405.592,-136.599,174.130,45.075,158.995
C02421=1039.162,405.346,-136.554,174.119,45.070,158.992
C02422=1039.152,405.101,-136.509,174.110,45.064,158.990
C02423=1039.142,404.855,-136.464,174.101,45.059,158.987
C02424=1039.132,404.609,-136.417,174.090,45.054,158.985
C02425=1039.123,404.364,-136.373,174.081,45.048,158.982
C02426=1039.113,404.118,-136.328,174.072,45.042,158.980
C02427=1039.104,403.873,-136.282,174.062,45.037,158.978
C02428=1039.094,403.627,-136.238,174.052,45.031,158.975
C02429=1039.085,403.381,-136.193,174.043,45.026,158.973
C02430=1039.075,403.135,-136.148,174.034,45.020,158.970
C02431=1039.065,402.889,-136.103,174.025,45.015,158.968
C02432=1039.056,402.643,-136.058,174.015,45.010,158.966
C02433=1039.046,402.398,-136.013,174.006,45.004,158.963
C02434=1039.037,402.152,-135.969,173.996,44.999,158.961
C02435=1039.027,401.906,-135.924,173.987,44.993,158.959
C02436=1039.017,401.661,-135.879,173.978,44.988,158.956
C02437=1039.008,401.415,-135.835,173.968,44.982,158.954
C02438=1038.998,401.169,-135.791,173.959,44.977,158.952
C02439=1038.989,400.923,-135.746,173.950,44.972,158.949
C02440=1038.979,400.677,-135.702,173.941,44.966,158.947
C02441=1038.970,400.431,-135.657,173.932,44.962,158.945
C02442=1038.960,400.186,-135.613,173.923,44.956,158.942
C02443=1038.951,399.940,-135.569,173.914,44.951,158.940
C02444=1038.942,399.694,-135.525,173.905,44.946,158.938
C02445=1038.932,399.449,-135.480,173.896,44.941,158.936
C02446=1038.923,399.202,-135.436,173.887,44.935,158.933
C02447=1038.913,398.956,-135.392,173.878,44.930,158.931
C02448=1038.903,398.711,-135.348,173.869,44.925,158.929
C02449=1038.894,398.465,-135.305,173.860,44.920,158.927
C02450=1038.885,398.219,-135.260,173.851,44.915,158.924
C02451=1038.875,397.973,-135.216,173.842,44.910,158.922
C02452=1038.866,397.727,-135.171,173.833,44.905,158.920
C02453=1038.857,397.482,-135.128,173.824,44.900,158.918
C02454=1038.847,397.236,-135.084,173.815,44.894,158.916
C02455=1038.837,396.990,-135.040,173.806,44.889,158.913
C02456=1038.829,396.744,-134.997,173.798,44.884,158.911
C02457=1038.819,396.498,-134.953,173.789,44.879,158.909
C02458=1038.810,396.252,-134.909,173.780,44.874,158.907
C02459=1038.801,396.006,-134.865,173.771,44.869,158.905
C02460=1038.792,395.760,-134.821,173.762,44.864,158.903
C02461=1038.783,395.514,-134.779,173.754,44.860,158.901
C02462=1038.773,395.268,-134.734,173.746,44.855,158.898
C02463=1038.764,395.023,-134.691,173.737,44.850,158.896
C02464=1038.755,394.776,-134.647,173.728,44.845,158.894
C02465=1038.746,394.531,-134.604,173.719,44.840,158.892
C02466=1038.737,394.284,-134.561,173.711,44.835,158.890
C02467=1038.727,394.039,-134.518,173.703,44.830,158.888
C02468=1038.718,393.792,-134.474,173.694,44.826,158.886
C02469=1038.709,393.547,-134.431,173.685,44.821,158.884
C02470=1038.699,393.300,-134.388,173.677,44.816,158.882
C02471=1038.690,393.055,-134.344,173.669,44.811,158.880
C02472=1038.683,392.840,-134.307,173.661,44.807,158.878
C02473=1038.675,392.626,-134.269,173.654,44.803,158.876
C02474=1038.667,392.411,-134.231,173.646,44.799,158.874
C02475=1038.659,392.197,-134.193,173.639,44.795,158.873
C02476=1038.651,391.983,-134.156,173.632,44.791,158.871
C02477=1038.643,391.768,-134.119,173.624,44.787,158.869
C02478=1038.635,391.554,-134.081,173.617,44.783,158.867
C02479=1038.628,391.339,-134.043,173.610,44.778,158.865
C02480=1038.618,391.094,-134.001,173.602,44.774,158.864
C02481=1038.610,390.848,-133.958,173.593,44.769,158.862
C02482=1038.600,390.601,-133.915,173.586,44.764,158.859
C02483=1038.591,390.355,-133.872,173.577,44.760,158.857
C02484=1038.582,390.109,-133.830,173.569,44.755,158.856
C02485=1038.574,389.863,-133.787,173.561,44.750,158.854
C02486=1038.564,389.617,-133.744,173.552,44.746,158.852
C02487=1038.556,389.370,-133.701,173.545,44.741,158.850
C02488=1038.546,389.124,-133.659,173.536,44.737,158.848
C02489=1038.538,388.878,-133.616,173.528,44.732,158.846
C02490=1038.529,388.633,-133.574,173.520,44.728,158.844
C02491=1038.520,388.387,-133.531,173.512,44.724,158.842
C02492=1038.511,388.140,-133.489,173.504,44.719,158.840
C02493=1038.502,387.894,-133.446,173.496,44.714,158.838
C02494=1038.493,387.647,-133.404,173.488,44.710,158.836
C02495=1038.484,387.401,-133.361,173.480,44.706,158.834
C02496=1038.475,387.155,-133.320,173.472,44.701,158.832
C02497=1038.466,386.909,-133.277,173.464,44.697,158.830
C02498=1038.458,386.663,-133.235,173.457,44.693,158.829
C02499=1038.448,386.417,-133.192,173.448,44.688,158.827
C02500=1038.439,386.170,-133.151,173.441,44.684,158.825
C02501=1038.431,385.924,-133.109,173.432,44.680,158.823
C02502=1038.421,385.678,-133.067,173.425,44.675,158.821
C02503=1038.413,385.432,-133.024,173.417,44.671,158.819
C02504=1038.404,385.185,-132.982,173.409,44.667,158.818
C02505=1038.395,384.940,-132.940,173.402,44.663,158.816
C02506=1038.386,384.693,-132.898,173.393,44.658,158.814
C02507=1038.377,384.447,-132.857,173.386,44.654,158.812
C02508=1038.368,384.200,-132.815,173.378,44.650,158.810
C02509=1038.360,383.954,-132.773,173.370,44.645,158.808
C02510=1038.352,383.708,-132.731,173.362,44.641,158.807
C02511=1038.343,383.462,-132.690,173.355,44.637,158.805
C02512=1038.334,383.215,-132.648,173.348,44.633,158.803
C02513=1038.325,382.969,-132.606,173.339,44.629,158.801
C02514=1038.317,382.722,-132.564,173.332,44.625,158.800
C02515=1038.308,382.477,-132.522,173.325,44.621,158.798
C02516=1038.299,382.230,-132.481,173.316,44.616,158.796
C02517=1038.290,381.984,-132.439,173.309,44.612,158.794
C02518=1038.281,381.738,-132.397,173.302,44.608,158.792
C02519=1038.273,381.492,-132.356,173.294,44.604,158.791
C02520=1038.265,381.245,-132.314,173.287,44.600,158.789
C02521=1038.256,380.998,-132.273,173.279,44.596,158.787
C02522=1038.248,380.753,-132.231,173.272,44.592,158.785
C02523=1038.239,380.506,-132.190,173.264,44.588,158.784
C02524=1038.230,380.259,-132.149,173.257,44.584,158.782
C02525=1038.222,380.014,-132.107,173.250,44.580,158.780
C02526=1038.213,379.767,-132.065,173.242,44.575,158.779
C02527=1038.205,379.520,-132.024,173.234,44.571,158.777
C02528=1038.197,379.274,-131.983,173.227,44.568,158.775
C02529=1038.188,379.027,-131.942,173.220,44.564,158.773
C02530=1038.180,378.782,-131.900,173.212,44.559,158.772
C02531=1038.171,378.535,-131.859,173.205,44.556,158.770
C02532=1038.158,378.140,-131.793,173.194,44.549,158.767
C02533=1038.144,377.746,-131.727,173.182,44.543,158.765
C02534=1038.130,377.351,-131.663,173.171,44.537,158.762
C02535=1038.117,376.957,-131.596,173.158,44.531,158.759
C02536=1038.109,376.711,-131.556,173.151,44.527,158.758
C02537=1038.099,376.464,-131.515,173.144,44.524,158.756
C02538=1038.091,376.218,-131.475,173.137,44.519,158.755
C02539=1038.083,375.972,-131.434,173.130,44.516,158.753
C02540=1038.075,375.725,-131.393,173.123,44.512,158.751
C02541=1038.066,375.478,-131.352,173.115,44.508,158.750
C02542=1038.057,375.232,-131.312,173.108,44.504,158.748
C02543=1038.049,374.985,-131.271,173.101,44.501,158.747
C02544=1038.041,374.739,-131.231,173.094,44.497,158.745
C02545=1038.032,374.492,-131.190,173.087,44.494,158.743
C02546=1038.024,374.246,-131.149,173.080,44.490,158.742
C02547=1038.015,373.999,-131.109,173.073,44.486,158.740
C02548=1038.007,373.753,-131.068,173.066,44.482,158.739
C02549=1037.999,373.507,-131.027,173.059,44.478,158.737
C02550=1037.991,373.260,-130.987,173.052,44.475,158.735
C02551=1037.983,373.013,-130.946,173.046,44.471,158.734
C02552=1037.974,372.767,-130.906,173.039,44.467,158.732
C02553=1037.966,372.520,-130.866,173.032,44.464,158.731
C02554=1037.958,372.274,-130.825,173.025,44.460,158.729
C02555=1037.950,372.027,-130.785,173.018,44.456,158.728
C02556=1037.941,371.780,-130.744,173.011,44.453,158.726
C02557=1037.933,371.534,-130.705,173.004,44.449,158.725
C02558=1037.925,371.287,-130.664,172.997,44.446,158.723
C02559=1037.917,371.041,-130.624,172.991,44.442,158.722
C02560=1037.909,370.794,-130.584,172.984,44.439,158.720
C02561=1037.900,370.547,-130.543,172.977,44.435,158.719
C02562=1037.892,370.301,-130.503,172.970,44.431,158.717
C02563=1037.884,370.054,-130.463,172.963,44.428,158.716
C02564=1037.876,369.808,-130.423,172.956,44.425,158.714
C02565=1037.868,369.561,-130.384,172.950,44.421,158.713
C02566=1037.859,369.315,-130.343,172.943,44.418,158.711
C02567=1037.851,369.068,-130.304,172.936,44.414,158.710
C02568=1037.843,368.821,-130.264,172.929,44.411,158.708
C02569=1037.835,368.574,-130.224,172.922,44.407,158.707
C02570=1037.826,368.327,-130.185,172.917,44.404,158.705
C02571=1037.817,368.081,-130.145,172.909,44.400,158.704
C02572=1037.810,367.834,-130.105,172.903,44.397,158.702
C02573=1037.801,367.588,-130.065,172.896,44.394,158.701
C02574=1037.794,367.341,-130.025,172.890,44.390,158.699
C02575=1037.785,367.094,-129.986,172.883,44.387,158.698
C02576=1037.777,366.847,-129.946,172.876,44.384,158.697
C02577=1037.769,366.601,-129.907,172.869,44.381,158.695
C02578=1037.761,366.354,-129.867,172.864,44.377,158.694
C02579=1037.753,366.107,-129.828,172.857,44.374,158.692
C02580=1037.744,365.861,-129.788,172.850,44.371,158.691
C02581=1037.737,365.614,-129.749,172.843,44.368,158.690
C02582=1037.729,365.368,-129.709,172.837,44.364,158.688
C02583=1037.721,365.121,-129.670,172.830,44.361,158.687
C02584=1037.713,364.874,-129.630,172.824,44.358,158.685
C02585=1037.705,364.627,-129.591,172.818,44.354,158.684
C02586=1037.697,364.380,-129.552,172.811,44.351,158.683
C02587=1037.688,364.134,-129.512,172.805,44.348,158.681
C02588=1037.681,363.876,-129.471,172.798,44.344,158.680
C02589=1037.672,363.619,-129.430,172.791,44.341,158.678
C02590=1037.664,363.362,-129.389,172.784,44.337,158.677
C02591=1037.655,363.105,-129.348,172.778,44.334,158.675
C02592=1037.649,362.871,-129.311,172.772,44.331,158.674
C02593=1037.641,362.637,-129.274,172.766,44.328,158.673
C02594=1037.633,362.390,-129.235,172.760,44.325,158.671
C02595=1037.625,362.143,-129.196,172.753,44.322,158.670
C02596=1037.617,361.897,-129.157,172.747,44.319,158.669
C02597=1037.609,361.649,-129.117,172.740,44.316,158.667
C02598=1037.601,361.403,-129.078,172.735,44.312,158.666
C02599=1037.593,361.156,-129.040,172.728,44.309,158.665
C02600=1037.585,360.909,-129.001,172.721,44.306,158.663
C02601=1037.577,360.663,-128.962,172.716,44.303,158.662
C02602=1037.569,360.415,-128.923,172.709,44.300,158.661
C02603=1037.562,360.169,-128.885,172.703,44.297,158.659
C02604=1037.553,359.922,-128.845,172.696,44.294,158.658
C02605=1037.545,359.675,-128.807,172.691,44.291,158.657
C02606=1037.538,359.428,-128.768,172.684,44.288,158.656
C02607=1037.530,359.181,-128.730,172.678,44.285,158.654
C02608=1037.521,358.934,-128.691,172.672,44.282,158.653
C02609=1037.514,358.688,-128.652,172.666,44.279,158.652
C02610=1037.505,358.441,-128.614,172.660,44.276,158.650
C02611=1037.498,358.194,-128.575,172.654,44.273,158.649
C02612=1037.490,357.947,-128.537,172.647,44.271,158.648
C02613=1037.483,357.700,-128.498,172.642,44.267,158.647
C02614=1037.475,357.453,-128.459,172.635,44.264,158.645
C02615=1037.467,357.206,-128.421,172.629,44.261,158.644
C02616=1037.459,356.959,-128.382,172.623,44.258,158.643
C02617=1037.451,356.712,-128.344,172.617,44.256,158.642
C02618=1037.443,356.465,-128.306,172.612,44.253,158.640
C02619=1037.435,356.218,-128.267,172.605,44.250,158.639
C02620=1037.428,355.972,-128.229,172.599,44.247,158.638
C02621=1037.420,355.724,-128.190,172.593,44.244,158.636
C02622=1037.412,355.477,-128.153,172.587,44.241,158.635
C02623=1037.405,355.231,-128.114,172.581,44.239,158.634
C02624=1037.397,354.984,-128.076,172.575,44.236,158.633
C02625=1037.388,354.737,-128.038,172.569,44.232,158.632
C02626=1037.380,354.490,-128.000,172.563,44.230,158.630
C02627=1037.373,354.243,-127.962,172.557,44.227,158.629
C02628=1037.365,353.996,-127.923,172.551,44.225,158.628
C02629=1037.358,353.749,-127.886,172.545,44.221,158.627
C02630=1037.350,353.502,-127.848,172.540,44.219,158.626
C02631=1037.342,353.255,-127.809,172.533,44.216,158.624
C02632=1037.335,353.008,-127.771,172.528,44.213,158.623
C02633=1037.326,352.761,-127.733,172.522,44.211,158.622
C02634=1037.318,352.514,-127.696,172.516,44.208,158.621
C02635=1037.311,352.267,-127.658,172.510,44.205,158.620
C02636=1037.304,352.020,-127.620,172.505,44.202,158.619
C02637=1037.295,351.773,-127.581,172.498,44.200,158.617
C02638=1037.288,351.526,-127.544,172.493,44.197,158.616
C02639=1037.281,351.279,-127.506,172.487,44.194,158.615
C02640=1037.272,351.032,-127.468,172.481,44.191,158.614
C02641=1037.265,350.785,-127.431,172.475,44.189,158.612
C02642=1037.257,350.538,-127.393,172.470,44.186,158.612
C02643=1037.250,350.291,-127.355,172.464,44.184,158.610
C02644=1037.242,350.043,-127.317,172.458,44.181,158.609
C02645=1037.234,349.797,-127.280,172.452,44.178,158.608
C02646=1037.224,349.428,-127.224,172.444,44.174,158.606
C02647=1037.212,349.061,-127.168,172.435,44.170,158.604
C02648=1037.201,348.692,-127.112,172.427,44.167,158.603
C02649=1037.189,348.324,-127.056,172.419,44.163,158.601
C02650=1037.181,348.078,-127.019,172.412,44.160,158.600
C02651=1037.174,347.830,-126.981,172.407,44.158,158.599
C02652=1037.165,347.583,-126.944,172.402,44.155,158.598
C02653=1037.158,347.336,-126.906,172.396,44.152,158.597
C02654=1037.151,347.089,-126.869,172.390,44.150,158.596
C02655=1037.143,346.842,-126.832,172.384,44.148,158.595
C02656=1037.136,346.595,-126.794,172.379,44.145,158.593
C02657=1037.128,346.348,-126.757,172.374,44.143,158.592
C02658=1037.120,346.101,-126.720,172.368,44.140,158.591
C02659=1037.113,345.854,-126.682,172.363,44.138,158.590
C02660=1037.105,345.606,-126.646,172.356,44.135,158.589
C02661=1037.098,345.359,-126.609,172.351,44.132,158.588
C02662=1037.090,345.112,-126.572,172.346,44.130,158.587
C02663=1037.083,344.865,-126.534,172.340,44.127,158.586
C02664=1037.075,344.618,-126.497,172.335,44.125,158.585
C02665=1037.068,344.371,-126.460,172.330,44.122,158.584
C02666=1037.060,344.124,-126.424,172.323,44.120,158.583
C02667=1037.053,343.877,-126.386,172.318,44.118,158.581
C02668=1037.045,343.630,-126.349,172.313,44.115,158.580
C02669=1037.038,343.382,-126.312,172.307,44.113,158.579
C02670=1037.030,343.135,-126.275,172.302,44.110,158.578
C02671=1037.023,342.887,-126.239,172.297,44.108,158.577
C02672=1037.015,342.641,-126.202,172.291,44.105,158.576
C02673=1037.008,342.393,-126.164,172.286,44.103,158.575
C02674=1037.000,342.146,-126.128,172.280,44.101,158.574
C02675=1036.993,341.899,-126.090,172.274,44.099,158.573
C02676=1036.985,341.651,-126.054,172.269,44.096,158.572
C02677=1036.978,341.404,-126.017,172.264,44.094,158.571
C02678=1036.971,341.158,-125.981,172.259,44.092,158.570
C02679=1036.963,340.911,-125.944,172.253,44.089,158.569
C02680=1036.956,340.663,-125.907,172.248,44.087,158.568
C02681=1036.948,340.416,-125.871,172.243,44.085,158.567
C02682=1036.940,340.169,-125.834,172.237,44.083,158.566
C02683=1036.933,339.921,-125.798,172.232,44.080,158.565
C02684=1036.926,339.673,-125.761,172.227,44.078,158.564
C02685=1036.919,339.427,-125.725,172.222,44.076,158.563
C02686=1036.911,339.180,-125.688,172.216,44.074,158.562
C02687=1036.903,338.932,-125.652,172.211,44.071,158.561
C02688=1036.896,338.685,-125.615,172.206,44.069,158.560
C02689=1036.888,338.437,-125.579,172.201,44.067,158.559
C02690=1036.881,338.191,-125.542,172.195,44.064,158.558
C02691=1036.873,337.944,-125.506,172.190,44.062,158.557
C02692=1036.866,337.696,-125.470,172.185,44.060,158.556
C02693=1036.859,337.448,-125.433,172.180,44.058,158.555
C02694=1036.852,337.202,-125.397,172.174,44.056,158.554
C02695=1036.844,336.954,-125.361,172.169,44.053,158.553
C02696=1036.836,336.707,-125.325,172.164,44.051,158.552
C02697=1036.829,336.459,-125.288,172.159,44.049,158.551
C02698=1036.822,336.212,-125.252,172.154,44.047,158.550
C02699=1036.815,335.965,-125.216,172.149,44.045,158.549
C02700=1036.807,335.718,-125.180,172.143,44.043,158.548
C02701=1036.800,335.471,-125.144,172.138,44.041,158.547
C02702=1036.789,335.099,-125.089,172.130,44.037,158.546
C02703=1036.778,334.727,-125.035,172.122,44.034,158.544
C02704=1036.767,334.356,-124.981,172.115,44.031,158.543
C02705=1036.756,333.984,-124.927,172.107,44.028,158.542
C02706=1036.749,333.737,-124.891,172.102,44.026,158.541
C02707=1036.741,333.490,-124.855,172.097,44.024,158.540
C02708=1036.734,333.242,-124.819,172.092,44.022,158.539
C02709=1036.727,332.995,-124.783,172.086,44.020,158.538
C02710=1036.719,332.748,-124.747,172.081,44.018,158.537
C02711=1036.712,332.500,-124.712,172.076,44.016,158.536
C02712=1036.705,332.253,-124.676,172.072,44.014,158.535
C02713=1036.697,332.006,-124.640,172.067,44.012,158.534
C02714=1036.689,331.758,-124.605,172.062,44.010,158.533
C02715=1036.682,331.511,-124.569,172.057,44.008,158.532
C02716=1036.675,331.264,-124.534,172.052,44.006,158.532
C02717=1036.667,331.016,-124.497,172.046,44.004,158.531
C02718=1036.660,330.769,-124.462,172.041,44.002,158.530
C02719=1036.653,330.522,-124.426,172.036,44.000,158.529
C02720=1036.646,330.275,-124.390,172.032,43.998,158.528
C02721=1036.639,330.027,-124.355,172.027,43.996,158.527
C02722=1036.632,329.779,-124.320,172.022,43.994,158.526
C02723=1036.624,329.532,-124.284,172.017,43.992,158.525
C02724=1036.617,329.284,-124.248,172.012,43.990,158.524
C02725=1036.610,329.038,-124.212,172.007,43.988,158.523
C02726=1036.603,328.790,-124.177,172.002,43.986,158.523
C02727=1036.596,328.543,-124.141,171.997,43.984,158.522
C02728=1036.588,328.296,-124.106,171.992,43.983,158.521
C02729=1036.581,328.048,-124.071,171.987,43.980,158.520
C02730=1036.573,327.801,-124.036,171.982,43.979,158.519
C02731=1036.566,327.553,-124.001,171.977,43.977,158.518
C02732=1036.559,327.306,-123.965,171.973,43.975,158.518
C02733=1036.551,327.058,-123.930,171.968,43.973,158.517
C02734=1036.544,326.811,-123.895,171.963,43.971,158.516
C02735=1036.536,326.564,-123.860,171.958,43.970,158.515
C02736=1036.529,326.316,-123.825,171.953,43.968,158.514
C02737=1036.522,326.069,-123.790,171.948,43.966,158.513
C02738=1036.515,325.821,-123.755,171.944,43.964,158.512
C02739=1036.507,325.573,-123.720,171.939,43.963,158.512
C02740=1036.500,325.326,-123.685,171.934,43.961,158.511
C02741=1036.492,325.079,-123.651,171.929,43.959,158.510
C02742=1036.485,324.831,-123.615,171.924,43.958,158.509
C02743=1036.477,324.584,-123.581,171.920,43.955,158.508
C02744=1036.471,324.336,-123.546,171.915,43.954,158.507
C02745=1036.463,324.089,-123.511,171.910,43.952,158.507
C02746=1036.456,323.841,-123.475,171.905,43.950,158.506
C02747=1036.448,323.594,-123.441,171.901,43.949,158.505
C02748=1036.442,323.347,-123.406,171.896,43.947,158.504
C02749=1036.433,323.099,-123.371,171.891,43.945,158.503
C02750=1036.427,322.851,-123.336,171.886,43.944,158.503
C02751=1036.419,322.604,-123.302,171.882,43.942,158.502
C02752=1036.413,322.357,-123.267,171.877,43.940,158.501
C02753=1036.405,322.109,-123.232,171.872,43.939,158.500
C02754=1036.398,321.862,-123.197,171.867,43.937,158.499
C02755=1036.391,321.614,-123.163,171.863,43.935,158.499
C02756=1036.384,321.367,-123.128,171.858,43.933,158.498
C02757=1036.376,321.120,-123.093,171.853,43.932,158.497
C02758=1036.365,320.743,-123.040,171.847,43.929,158.496
C02759=1036.355,320.367,-122.988,171.839,43.927,158.495
C02760=1036.343,319.991,-122.935,171.832,43.924,158.493
C02761=1036.333,319.615,-122.883,171.825,43.922,158.492
C02762=1036.326,319.367,-122.848,171.820,43.920,158.491
C02763=1036.318,319.119,-122.813,171.816,43.918,158.491
C02764=1036.311,318.872,-122.778,171.811,43.916,158.490
C02765=1036.304,318.624,-122.745,171.806,43.915,158.489
C02766=1036.298,318.377,-122.709,171.802,43.913,158.488
C02767=1036.290,318.129,-122.676,171.797,43.911,158.487
C02768=1036.284,317.882,-122.640,171.793,43.910,158.487
C02769=1036.276,317.634,-122.607,171.789,43.909,158.486
C02770=1036.270,317.387,-122.571,171.784,43.907,158.485
C02771=1036.262,317.139,-122.538,171.779,43.905,158.484
C02772=1036.256,316.892,-122.502,171.775,43.903,158.484
C02773=1036.248,316.644,-122.469,171.770,43.902,158.483
C02774=1036.241,316.397,-122.435,171.766,43.900,158.482
C02775=1036.234,316.149,-122.400,171.761,43.899,158.481
C02776=1036.227,315.902,-122.366,171.756,43.897,158.481
C02777=1036.221,315.655,-122.331,171.752,43.895,158.480
C02778=1036.214,315.407,-122.297,171.748,43.894,158.479
C02779=1036.207,315.159,-122.263,171.744,43.892,158.478
C02780=1036.200,314.912,-122.228,171.739,43.891,158.478
C02781=1036.193,314.665,-122.195,171.735,43.889,158.477
C02782=1036.186,314.417,-122.160,171.730,43.888,158.476
C02783=1036.179,314.169,-122.126,171.725,43.886,158.475
C02784=1036.172,313.922,-122.091,171.721,43.884,158.475
C02785=1036.166,313.675,-122.058,171.716,43.883,158.474
C02786=1036.158,313.427,-122.024,171.712,43.882,158.473
C02787=1036.152,313.179,-121.989,171.707,43.880,158.472
C02788=1036.145,312.932,-121.955,171.703,43.878,158.472
C02789=1036.138,312.684,-121.920,171.699,43.877,158.471
C02790=1036.131,312.437,-121.887,171.695,43.875,158.470
C02791=1036.125,312.189,-121.853,171.690,43.874,158.470
C02792=1036.117,311.942,-121.818,171.686,43.872,158.469
C02793=1036.110,311.694,-121.784,171.681,43.871,158.468
C02794=1036.103,311.446,-121.750,171.677,43.869,158.467
C02795=1036.096,311.198,-121.717,171.673,43.868,158.467
C02796=1036.090,310.951,-121.684,171.668,43.867,158.466
C02797=1036.082,310.704,-121.650,171.664,43.865,158.465
C02798=1036.074,310.456,-121.617,171.659,43.864,158.464
C02799=1036.067,310.209,-121.583,171.655,43.863,158.464
C02800=1036.060,309.961,-121.549,171.650,43.861,158.463
C02801=1036.053,309.714,-121.516,171.646,43.860,158.462
C02802=1036.047,309.466,-121.483,171.642,43.859,158.462
C02803=1036.039,309.218,-121.449,171.638,43.857,158.461
C02804=1036.031,308.971,-121.416,171.633,43.856,158.460
C02805=1036.024,308.723,-121.382,171.628,43.855,158.460
C02806=1036.018,308.475,-121.349,171.625,43.853,158.459
C02807=1036.011,308.228,-121.315,171.620,43.852,158.459
C02808=1036.004,307.980,-121.281,171.616,43.850,158.458
C02809=1035.996,307.733,-121.248,171.611,43.849,158.457
C02810=1035.989,307.485,-121.215,171.607,43.848,158.457
C02811=1035.982,307.237,-121.181,171.603,43.847,158.456
C02812=1035.975,306.990,-121.148,171.599,43.845,158.455
C02813=1035.969,306.742,-121.115,171.594,43.844,158.454
C02814=1035.958,306.371,-121.065,171.588,43.842,158.453
C02815=1035.947,305.999,-121.015,171.582,43.840,158.452
C02816=1035.936,305.628,-120.965,171.576,43.839,158.452
C02817=1035.926,305.257,-120.915,171.569,43.837,158.451
C02818=1035.919,305.008,-120.882,171.565,43.835,158.450
C02819=1035.912,304.761,-120.849,171.561,43.834,158.449
C02820=1035.905,304.513,-120.816,171.556,43.833,158.449
C02821=1035.897,304.266,-120.782,171.552,43.831,158.448
C02822=1035.891,304.018,-120.750,171.548,43.830,158.447
C02823=1035.884,303.771,-120.716,171.544,43.829,158.447
C02824=1035.878,303.523,-120.683,171.540,43.828,158.446
C02825=1035.870,303.276,-120.650,171.535,43.827,158.445
C02826=1035.863,303.027,-120.617,171.532,43.825,158.445
C02827=1035.856,302.780,-120.584,171.527,43.824,158.444
C02828=1035.849,302.532,-120.550,171.523,43.823,158.443
C02829=1035.843,302.284,-120.517,171.519,43.821,158.443
C02830=1035.835,302.037,-120.484,171.514,43.820,158.442
C02831=1035.829,301.790,-120.451,171.511,43.819,158.442
C02832=1035.822,301.541,-120.418,171.506,43.818,158.441
C02833=1035.815,301.294,-120.385,171.502,43.817,158.440
C02834=1035.808,301.046,-120.352,171.499,43.815,158.440
C02835=1035.801,300.799,-120.320,171.494,43.814,158.439
C02836=1035.794,300.550,-120.287,171.490,43.813,158.438
C02837=1035.788,300.303,-120.253,171.485,43.812,158.438
C02838=1035.780,300.055,-120.221,171.482,43.811,158.437
C02839=1035.774,299.808,-120.188,171.478,43.809,158.437
C02840=1035.768,299.560,-120.155,171.473,43.808,158.436
C02841=1035.761,299.312,-120.122,171.469,43.807,158.435
C02842=1035.753,299.065,-120.089,171.466,43.806,158.435
C02843=1035.747,298.817,-120.056,171.461,43.805,158.434
C02844=1035.740,298.569,-120.023,171.457,43.804,158.434
C02845=1035.734,298.322,-119.991,171.454,43.802,158.433
C02846=1035.726,298.074,-119.958,171.449,43.801,158.432
C02847=1035.720,297.826,-119.925,171.445,43.800,158.432
C02848=1035.713,297.578,-119.892,171.441,43.799,158.431
C02849=1035.707,297.330,-119.859,171.438,43.797,158.430
C02850=1035.700,297.083,-119.827,171.433,43.796,158.430
C02851=1035.693,296.835,-119.793,171.429,43.795,158.429
C02852=1035.686,296.588,-119.761,171.426,43.794,158.429
C02853=1035.680,296.340,-119.728,171.421,43.793,158.428
C02854=1035.672,296.092,-119.695,171.417,43.792,158.427
C02855=1035.666,295.845,-119.663,171.414,43.791,158.427
C02856=1035.660,295.597,-119.630,171.410,43.790,158.426
C02857=1035.653,295.349,-119.599,171.405,43.789,158.426
C02858=1035.646,295.101,-119.565,171.401,43.787,158.425
C02859=1035.640,294.853,-119.533,171.398,43.786,158.425
C02860=1035.633,294.606,-119.501,171.393,43.785,158.424
C02861=1035.626,294.358,-119.467,171.389,43.784,158.423
C02862=1035.619,294.110,-119.435,171.386,43.783,158.423
C02863=1035.612,293.862,-119.404,171.382,43.782,158.422
C02864=1035.605,293.614,-119.371,171.377,43.781,158.422
C02865=1035.598,293.367,-119.339,171.374,43.780,158.421
C02866=1035.592,293.119,-119.306,171.370,43.779,158.421
C02867=1035.585,292.871,-119.274,171.365,43.778,158.420
C02868=1035.578,292.623,-119.242,171.362,43.777,158.419
C02869=1035.571,292.376,-119.209,171.358,43.776,158.419
C02870=1035.562,292.021,-119.164,171.352,43.774,158.418
C02871=1035.552,291.667,-119.117,171.347,43.773,158.417
C02872=1035.541,291.311,-119.071,171.341,43.772,158.417
C02873=1035.532,290.957,-119.026,171.336,43.770,158.416
C02874=1035.525,290.709,-118.993,171.332,43.769,158.415
C02875=1035.518,290.462,-118.962,171.328,43.768,158.415
C02876=1035.512,290.214,-118.929,171.325,43.767,158.414
C02877=1035.505,289.966,-118.898,171.320,43.767,158.414
C02878=1035.497,289.718,-118.865,171.316,43.765,158.413
C02879=1035.491,289.470,-118.834,171.313,43.764,158.412
C02880=1035.484,289.223,-118.801,171.309,43.763,158.412
C02881=1035.478,288.975,-118.770,171.304,43.762,158.411
C02882=1035.471,288.727,-118.738,171.301,43.762,158.411
C02883=1035.463,288.479,-118.706,171.297,43.760,158.410
C02884=1035.456,288.232,-118.674,171.294,43.760,158.410
C02885=1035.450,287.983,-118.642,171.290,43.759,158.409
C02886=1035.444,287.735,-118.610,171.286,43.758,158.409
C02887=1035.437,287.488,-118.578,171.282,43.757,158.408
C02888=1035.430,287.240,-118.547,171.278,43.756,158.408
C02889=1035.422,286.992,-118.515,171.275,43.755,158.407
C02890=1035.415,286.744,-118.483,171.271,43.754,158.407
C02891=1035.409,286.496,-118.451,171.266,43.753,158.406
C02892=1035.403,286.248,-118.419,171.263,43.752,158.406
C02893=1035.396,286.000,-118.388,171.259,43.752,158.405
C02894=1035.389,285.752,-118.356,171.256,43.751,158.404
C02895=1035.382,285.505,-118.324,171.252,43.750,158.404
C02896=1035.376,285.257,-118.293,171.249,43.749,158.404
C02897=1035.367,285.009,-118.262,171.244,43.748,158.403
C02898=1035.361,284.761,-118.230,171.240,43.747,158.403
C02899=1035.354,284.513,-118.199,171.237,43.747,158.402
C02900=1035.347,284.265,-118.167,171.233,43.746,158.401
C02901=1035.341,284.017,-118.136,171.230,43.745,158.401
C02902=1035.334,283.769,-118.104,171.225,43.744,158.401
C02903=1035.327,283.522,-118.072,171.222,43.743,158.400
C02904=1035.320,283.274,-118.041,171.218,43.742,158.400
C02905=1035.313,283.026,-118.009,171.215,43.742,158.399
C02906=1035.307,282.778,-117.978,171.211,43.741,158.398
C02907=1035.300,282.531,-117.947,171.207,43.740,158.398
C02908=1035.293,282.283,-117.915,171.204,43.739,158.398
C02909=1035.286,282.035,-117.884,171.199,43.738,158.397
C02910=1035.280,281.787,-117.852,171.196,43.737,158.397
C02911=1035.273,281.539,-117.821,171.192,43.737,158.396
C02912=1035.266,281.291,-117.789,171.189,43.736,158.396
C02913=1035.260,281.043,-117.758,171.185,43.735,158.395
C02914=1035.253,280.795,-117.727,171.182,43.734,158.395
C02915=1035.246,280.547,-117.696,171.178,43.734,158.394
C02916=1035.240,280.299,-117.664,171.175,43.733,158.394
C02917=1035.233,280.051,-117.633,171.171,43.732,158.393
C02918=1035.226,279.803,-117.601,171.167,43.731,158.393
C02919=1035.219,279.555,-117.570,171.163,43.730,158.392
C02920=1035.213,279.307,-117.539,171.159,43.730,158.392
C02921=1035.205,279.060,-117.508,171.156,43.729,158.391
C02922=1035.199,278.811,-117.477,171.152,43.728,158.391
C02923=1035.192,278.563,-117.446,171.149,43.727,158.390
C02924=1035.185,278.315,-117.414,171.145,43.727,158.390
C02925=1035.179,278.067,-117.383,171.142,43.726,158.389
C02926=1035.170,277.724,-117.340,171.137,43.725,158.389
C02927=1035.160,277.382,-117.298,171.131,43.724,158.388
C02928=1035.151,277.040,-117.255,171.127,43.723,158.387
C02929=1035.142,276.697,-117.212,171.122,43.722,158.387
C02930=1035.135,276.449,-117.180,171.118,43.721,158.386
C02931=1035.128,276.201,-117.150,171.115,43.720,158.386
C02932=1035.121,275.953,-117.119,171.111,43.720,158.385
C02933=1035.115,275.705,-117.088,171.108,43.719,158.385
C02934=1035.107,275.457,-117.057,171.104,43.718,158.385
C02935=1035.101,275.209,-117.026,171.101,43.717,158.384
C02936=1035.095,274.961,-116.995,171.097,43.716,158.384
C02937=1035.087,274.714,-116.965,171.094,43.716,158.383
C02938=1035.081,274.465,-116.934,171.090,43.715,158.383
C02939=1035.074,274.217,-116.902,171.086,43.715,158.382
C02940=1035.067,273.969,-116.872,171.082,43.714,158.382
C02941=1035.060,273.721,-116.841,171.079,43.713,158.381
C02942=1035.054,273.473,-116.810,171.075,43.713,158.381
C02943=1035.047,273.225,-116.780,171.072,43.712,158.380
C02944=1035.041,272.977,-116.749,171.068,43.711,158.380
C02945=1035.034,272.729,-116.718,171.065,43.711,158.380
C02946=1035.027,272.481,-116.687,171.061,43.710,158.379
C02947=1035.020,272.233,-116.657,171.058,43.709,158.379
C02948=1035.013,271.986,-116.626,171.054,43.709,158.378
C02949=1035.007,271.737,-116.596,171.051,43.708,158.378
C02950=1035.001,271.489,-116.565,171.047,43.707,158.377
C02951=1034.993,271.241,-116.534,171.044,43.707,158.377
C02952=1034.987,270.993,-116.504,171.040,43.706,158.376
C02953=1034.980,270.745,-116.474,171.037,43.706,158.376
C02954=1034.974,270.497,-116.443,171.034,43.705,158.376
C02955=1034.966,270.249,-116.412,171.030,43.705,158.375
C02956=1034.960,270.001,-116.382,171.027,43.704,158.375
C02957=1034.953,269.753,-116.351,171.023,43.703,158.374
C02958=1034.946,269.505,-116.321,171.020,43.703,158.374
C02959=1034.939,269.257,-116.290,171.016,43.702,158.374
C02960=1034.933,269.009,-116.260,171.013,43.701,158.373
C02961=1034.926,268.761,-116.229,171.009,43.701,158.373
C02962=1034.919,268.513,-116.199,171.006,43.701,158.372
C02963=1034.913,268.264,-116.169,171.003,43.700,158.372
C02964=1034.906,268.017,-116.139,171.000,43.699,158.372
C02965=1034.899,267.768,-116.109,170.996,43.698,158.371
C02966=1034.892,267.520,-116.077,170.993,43.698,158.371
C02967=1034.886,267.273,-116.048,170.990,43.697,158.370
C02968=1034.879,267.024,-116.017,170.986,43.697,158.370
C02969=1034.872,266.776,-115.987,170.983,43.696,158.369
C02970=1034.866,266.529,-115.957,170.979,43.696,158.369
C02971=1034.859,266.280,-115.926,170.976,43.695,158.369
C02972=1034.852,266.032,-115.896,170.973,43.695,158.368
C02973=1034.845,265.784,-115.866,170.969,43.694,158.368
C02974=1034.839,265.536,-115.836,170.966,43.694,158.367
C02975=1034.832,265.288,-115.806,170.962,43.693,158.367
C02976=1034.825,265.040,-115.776,170.959,43.693,158.367
C02977=1034.818,264.792,-115.746,170.955,43.692,158.366
C02978=1034.812,264.543,-115.716,170.952,43.691,158.366
C02979=1034.806,264.295,-115.686,170.948,43.691,158.365
C02980=1034.798,264.047,-115.656,170.945,43.691,158.365
C02981=1034.791,263.799,-115.626,170.943,43.690,158.365
C02982=1034.783,263.461,-115.584,170.938,43.689,158.364
C02983=1034.773,263.123,-115.544,170.933,43.688,158.364
C02984=1034.764,262.785,-115.503,170.929,43.688,158.363
C02985=1034.756,262.448,-115.462,170.924,43.687,158.363
C02986=1034.749,262.199,-115.432,170.921,43.687,158.362
C02987=1034.742,261.951,-115.402,170.917,43.686,158.362
C02988=1034.735,261.704,-115.372,170.914,43.685,158.361
C02989=1034.729,261.454,-115.342,170.911,43.685,158.361
C02990=1034.723,261.207,-115.312,170.907,43.685,158.361
C02991=1034.715,260.959,-115.283,170.904,43.684,158.360
C02992=1034.708,260.710,-115.253,170.900,43.684,158.360
C02993=1034.701,260.463,-115.223,170.897,43.684,158.360
C02994=1034.694,260.214,-115.194,170.895,43.683,158.359
C02995=1034.688,259.966,-115.164,170.891,43.683,158.359
C02996=1034.681,259.718,-115.134,170.888,43.682,158.358
C02997=1034.674,259.469,-115.105,170.885,43.682,158.358
C02998=1034.667,259.222,-115.075,170.881,43.681,158.358
C02999=1034.660,258.973,-115.046,170.878,43.681,158.357
C03000=1034.653,258.726,-115.016,170.875,43.681,158.357
C03001=1034.646,258.477,-114.987,170.871,43.681,158.357
C03002=1034.640,258.229,-114.957,170.868,43.680,158.356
C03003=1034.633,257.981,-114.928,170.865,43.680,158.356
C03004=1034.626,257.732,-114.898,170.862,43.679,158.356
C03005=1034.619,257.484,-114.869,170.859,43.679,158.355
C03006=1034.612,257.236,-114.839,170.855,43.678,158.355
C03007=1034.605,256.988,-114.810,170.852,43.678,158.355
C03008=1034.598,256.740,-114.780,170.849,43.678,158.354
C03009=1034.592,256.492,-114.751,170.845,43.678,158.354
C03010=1034.585,256.243,-114.722,170.842,43.677,158.353
C03011=1034.578,255.996,-114.692,170.840,43.677,158.353
C03012=1034.572,255.747,-114.662,170.836,43.676,158.353
C03013=1034.565,255.499,-114.633,170.833,43.676,158.352
C03014=1034.557,255.251,-114.604,170.830,43.676,158.352
C03015=1034.551,255.003,-114.575,170.826,43.675,158.352
C03016=1034.545,254.755,-114.545,170.823,43.675,158.351
C03017=1034.538,254.506,-114.516,170.820,43.674,158.351
C03018=1034.532,254.258,-114.487,170.817,43.674,158.351
C03019=1034.524,254.010,-114.457,170.814,43.673,158.350
C03020=1034.518,253.762,-114.427,170.810,43.673,158.350
C03021=1034.511,253.513,-114.399,170.807,43.673,158.350
C03022=1034.504,253.266,-114.369,170.804,43.673,158.349
C03023=1034.498,253.018,-114.340,170.801,43.672,158.349
C03024=1034.491,252.769,-114.310,170.798,43.672,158.349
C03025=1034.485,252.521,-114.281,170.795,43.672,158.348
C03026=1034.478,252.272,-114.251,170.791,43.671,158.348
C03027=1034.471,252.024,-114.222,170.788,43.671,158.348
C03028=1034.464,251.776,-114.194,170.785,43.670,158.347
C03029=1034.457,251.528,-114.164,170.782,43.670,158.347
C03030=1034.451,251.279,-114.135,170.779,43.670,158.347
C03031=1034.445,251.032,-114.106,170.775,43.669,158.346
C03032=1034.438,250.783,-114.076,170.773,43.669,158.346
C03033=1034.432,250.535,-114.047,170.770,43.668,158.346
C03034=1034.425,250.287,-114.019,170.766,43.668,158.345
C03035=1034.418,250.038,-113.989,170.763,43.668,158.345
C03036=1034.411,249.790,-113.960,170.761,43.667,158.345
C03037=1034.405,249.542,-113.931,170.757,43.667,158.344
C03038=1034.396,249.203,-113.891,170.753,43.667,158.344
C03039=1034.387,248.864,-113.852,170.748,43.666,158.343
C03040=1034.378,248.524,-113.812,170.745,43.666,158.343
C03041=1034.368,248.185,-113.772,170.740,43.665,158.342
C03042=1034.362,247.937,-113.742,170.737,43.665,158.342
C03043=1034.355,247.688,-113.713,170.734,43.664,158.342
C03044=1034.349,247.440,-113.684,170.731,43.664,158.341
C03045=1034.343,247.192,-113.655,170.728,43.664,158.341
C03046=1034.336,246.943,-113.626,170.725,43.663,158.341
C03047=1034.329,246.696,-113.598,170.722,43.663,158.340
C03048=1034.323,246.447,-113.568,170.719,43.663,158.340
C03049=1034.317,246.199,-113.539,170.716,43.662,158.340
C03050=1034.310,245.950,-113.510,170.712,43.662,158.339
C03051=1034.303,245.702,-113.481,170.710,43.661,158.339
C03052=1034.296,245.454,-113.453,170.707,43.661,158.339
C03053=1034.290,245.206,-113.423,170.703,43.661,158.338
C03054=1034.284,244.958,-113.394,170.701,43.661,158.338
C03055=1034.277,244.709,-113.366,170.698,43.660,158.338
C03056=1034.270,244.461,-113.337,170.694,43.660,158.338
C03057=1034.264,244.213,-113.308,170.692,43.660,158.337
C03058=1034.257,243.965,-113.280,170.689,43.659,158.337
C03059=1034.251,243.717,-113.251,170.685,43.659,158.337
C03060=1034.244,243.467,-113.222,170.682,43.659,158.336
C03061=1034.237,243.220,-113.194,170.680,43.659,158.336
C03062=1034.231,242.971,-113.165,170.676,43.658,158.336
C03063=1034.224,242.724,-113.136,170.673,43.658,158.335
C03064=1034.217,242.475,-113.107,170.671,43.658,158.335
C03065=1034.211,242.226,-113.079,170.668,43.658,158.335
C03066=1034.204,241.978,-113.050,170.664,43.657,158.334
C03067=1034.197,241.730,-113.022,170.662,43.657,158.334
C03068=1034.191,241.482,-112.993,170.659,43.657,158.334
C03069=1034.184,241.234,-112.965,170.655,43.657,158.334
C03070=1034.178,240.985,-112.935,170.653,43.657,158.333
C03071=1034.171,240.737,-112.908,170.650,43.656,158.333
C03072=1034.165,240.488,-112.879,170.646,43.656,158.333
C03073=1034.158,240.241,-112.850,170.644,43.656,158.332
C03074=1034.152,239.992,-112.822,170.641,43.656,158.332
C03075=1034.145,239.744,-112.793,170.638,43.656,158.332
C03076=1034.138,239.496,-112.766,170.635,43.655,158.331
C03077=1034.131,239.247,-112.737,170.632,43.655,158.331
C03078=1034.125,238.998,-112.709,170.629,43.655,158.331
C03079=1034.118,238.750,-112.680,170.627,43.655,158.331
C03080=1034.111,238.502,-112.652,170.623,43.654,158.330
C03081=1034.105,238.254,-112.623,170.620,43.654,158.330
C03082=1034.098,238.005,-112.596,170.618,43.654,158.330
C03083=1034.091,237.758,-112.567,170.614,43.654,158.329
C03084=1034.084,237.509,-112.539,170.611,43.654,158.329
C03085=1034.077,237.260,-112.510,170.609,43.654,158.329
C03086=1034.071,237.012,-112.482,170.606,43.654,158.329
C03087=1034.064,236.764,-112.454,170.602,43.653,158.328
C03088=1034.057,236.516,-112.426,170.600,43.653,158.328
C03089=1034.051,236.267,-112.398,170.597,43.653,158.328
C03090=1034.044,236.019,-112.369,170.594,43.653,158.328
C03091=1034.037,235.771,-112.342,170.591,43.653,158.327
C03092=1034.031,235.522,-112.314,170.588,43.653,158.327
C03093=1034.024,235.274,-112.285,170.586,43.653,158.327
C03094=1034.015,234.929,-112.246,170.581,43.652,158.326
C03095=1034.005,234.583,-112.207,170.577,43.652,158.326
C03096=1033.997,234.238,-112.168,170.574,43.651,158.325
C03097=1033.987,233.892,-112.129,170.569,43.652,158.325
C03098=1033.980,233.645,-112.101,170.566,43.652,158.325
C03099=1033.973,233.396,-112.073,170.564,43.651,158.325
C03100=1033.967,233.147,-112.045,170.561,43.651,158.324
C03101=1033.960,232.900,-112.016,170.558,43.651,158.324
C03102=1033.954,232.651,-111.988,170.555,43.651,158.324
C03103=1033.947,232.403,-111.961,170.552,43.651,158.324
C03104=1033.940,232.154,-111.933,170.550,43.651,158.323
C03105=1033.934,231.906,-111.905,170.546,43.651,158.323
C03106=1033.927,231.658,-111.876,170.544,43.650,158.323
C03107=1033.921,231.409,-111.849,170.541,43.650,158.322
C03108=1033.914,231.161,-111.821,170.539,43.650,158.322
C03109=1033.907,230.912,-111.793,170.535,43.650,158.322
C03110=1033.901,230.664,-111.765,170.532,43.650,158.322
C03111=1033.894,230.416,-111.738,170.530,43.650,158.321
C03112=1033.887,230.167,-111.710,170.526,43.649,158.321
C03113=1033.880,229.919,-111.681,170.524,43.649,158.321
C03114=1033.874,229.671,-111.654,170.521,43.649,158.321
C03115=1033.867,229.422,-111.626,170.518,43.649,158.320
C03116=1033.860,229.174,-111.598,170.515,43.649,158.320
C03117=1033.854,228.925,-111.570,170.512,43.649,158.320
C03118=1033.848,228.677,-111.542,170.510,43.649,158.320
C03119=1033.841,228.428,-111.514,170.507,43.648,158.319
C03120=1033.835,228.181,-111.487,170.504,43.648,158.319
C03121=1033.828,227.932,-111.459,170.501,43.648,158.319
C03122=1033.821,227.684,-111.432,170.499,43.648,158.319
C03123=1033.814,227.436,-111.404,170.496,43.648,158.318
C03124=1033.807,227.187,-111.377,170.493,43.648,158.318
C03125=1033.801,226.939,-111.349,170.490,43.648,158.318
C03126=1033.794,226.690,-111.321,170.487,43.648,158.318
C03127=1033.787,226.442,-111.294,170.485,43.648,158.317
C03128=1033.780,226.193,-111.267,170.482,43.648,158.317
C03129=1033.774,225.945,-111.239,170.479,43.648,158.317
C03130=1033.767,225.696,-111.212,170.476,43.648,158.317
C03131=1033.760,225.448,-111.184,170.474,43.648,158.316
C03132=1033.753,225.199,-111.156,170.471,43.648,158.316
C03133=1033.746,224.951,-111.129,170.468,43.648,158.316
C03134=1033.739,224.703,-111.101,170.465,43.647,158.316
C03135=1033.734,224.454,-111.075,170.462,43.647,158.315
C03136=1033.727,224.206,-111.047,170.460,43.648,158.315
C03137=1033.720,223.957,-111.019,170.457,43.648,158.315
C03138=1033.714,223.709,-110.992,170.455,43.647,158.315
C03139=1033.706,223.461,-110.964,170.451,43.647,158.314
C03140=1033.700,223.212,-110.937,170.449,43.647,158.314
C03141=1033.693,222.963,-110.910,170.446,43.647,158.314
C03142=1033.687,222.716,-110.882,170.444,43.647,158.314
C03143=1033.680,222.467,-110.855,170.440,43.647,158.314
C03144=1033.673,222.218,-110.828,170.438,43.647,158.313
C03145=1033.667,221.970,-110.800,170.435,43.647,158.313
C03146=1033.660,221.722,-110.773,170.433,43.647,158.313
C03147=1033.653,221.473,-110.746,170.429,43.647,158.312
C03148=1033.647,221.225,-110.719,170.427,43.647,158.312
C03149=1033.640,220.977,-110.691,170.424,43.647,158.312
C03150=1033.631,220.624,-110.652,170.421,43.647,158.312
C03151=1033.621,220.271,-110.614,170.416,43.646,158.311
C03152=1033.612,219.918,-110.574,170.413,43.646,158.311
C03153=1033.602,219.565,-110.536,170.409,43.646,158.311
C03154=1033.596,219.316,-110.509,170.407,43.646,158.310
C03155=1033.588,219.068,-110.482,170.404,43.647,158.310
C03156=1033.582,218.820,-110.455,170.401,43.647,158.310
C03157=1033.575,218.572,-110.428,170.398,43.646,158.310
C03158=1033.569,218.323,-110.400,170.396,43.647,158.310
C03159=1033.561,218.074,-110.374,170.393,43.647,158.309
C03160=1033.555,217.826,-110.346,170.391,43.647,158.309
C03161=1033.548,217.578,-110.320,170.387,43.646,158.309
C03162=1033.542,217.330,-110.292,170.385,43.647,158.309
C03163=1033.534,217.081,-110.266,170.382,43.647,158.309
C03164=1033.528,216.832,-110.239,170.380,43.646,158.308
C03165=1033.522,216.584,-110.212,170.377,43.647,158.308
C03166=1033.515,216.335,-110.185,170.374,43.647,158.308
C03167=1033.508,216.087,-110.157,170.372,43.647,158.308
C03168=1033.501,215.838,-110.131,170.369,43.647,158.308
C03169=1033.495,215.590,-110.104,170.367,43.647,158.307
C03170=1033.488,215.342,-110.077,170.364,43.647,158.307
C03171=1033.482,215.092,-110.050,170.362,43.647,158.307
C03172=1033.474,214.844,-110.023,170.358,43.647,158.307
C03173=1033.468,214.596,-109.996,170.356,43.647,158.306
C03174=1033.461,214.348,-109.969,170.353,43.647,158.306
C03175=1033.455,214.099,-109.942,170.351,43.647,158.306
C03176=1033.448,213.851,-109.916,170.349,43.647,158.306
C03177=1033.441,213.602,-109.889,170.345,43.647,158.305
C03178=1033.434,213.354,-109.862,170.343,43.647,158.305
C03179=1033.428,213.104,-109.835,170.340,43.647,158.305
C03180=1033.421,212.857,-109.808,170.338,43.647,158.305
C03181=1033.415,212.608,-109.781,170.336,43.647,158.305
C03182=1033.408,212.359,-109.755,170.333,43.647,158.304
C03183=1033.401,212.112,-109.728,170.330,43.647,158.304
C03184=1033.394,211.863,-109.701,170.327,43.647,158.304
C03185=1033.389,211.614,-109.674,170.325,43.647,158.304
C03186=1033.381,211.366,-109.648,170.323,43.647,158.304
C03187=1033.374,211.118,-109.621,170.319,43.647,158.303
C03188=1033.368,210.869,-109.594,170.317,43.647,158.303
C03189=1033.361,210.620,-109.568,170.314,43.647,158.303
C03190=1033.354,210.372,-109.541,170.312,43.648,158.303
C03191=1033.348,210.123,-109.515,170.310,43.647,158.303
C03192=1033.341,209.875,-109.488,170.307,43.647,158.302
C03193=1033.334,209.626,-109.461,170.305,43.648,158.302
C03194=1033.328,209.378,-109.435,170.301,43.648,158.302
C03195=1033.321,209.129,-109.408,170.299,43.648,158.302
C03196=1033.314,208.881,-109.382,170.297,43.648,158.302
C03197=1033.308,208.632,-109.355,170.294,43.648,158.301
C03198=1033.301,208.383,-109.329,170.292,43.648,158.301
C03199=1033.294,208.135,-109.303,170.289,43.648,158.301
C03200=1033.287,207.887,-109.276,170.287,43.648,158.301
C03201=1033.281,207.638,-109.248,170.284,43.648,158.301
C03202=1033.274,207.390,-109.222,170.281,43.648,158.300
C03203=1033.267,207.141,-109.196,170.279,43.648,158.300
C03204=1033.260,206.893,-109.170,170.276,43.648,158.300
C03205=1033.253,206.645,-109.144,170.274,43.649,158.300
C03206=1033.244,206.297,-109.107,170.270,43.649,158.300
C03207=1033.235,205.951,-109.070,170.266,43.649,158.299
C03208=1033.225,205.603,-109.033,170.263,43.649,158.299
C03209=1033.216,205.256,-108.997,170.260,43.649,158.299
C03210=1033.190,204.206,-108.891,169.924,43.545,158.249
C03211=1033.184,203.958,-108.866,169.921,43.546,158.249
C03212=1033.177,203.709,-108.841,169.917,43.546,158.249
C03213=1033.172,203.461,-108.816,169.914,43.547,158.249
C03214=1033.166,203.212,-108.791,169.910,43.548,158.249
C03215=1033.160,202.963,-108.766,169.907,43.549,158.249
C03216=1033.153,202.714,-108.740,169.903,43.550,158.249
C03217=1033.147,202.465,-108.716,169.900,43.551,158.249
C03218=1033.141,202.217,-108.691,169.896,43.552,158.249
C03219=1033.135,201.969,-108.666,169.893,43.552,158.248
C03220=1033.129,201.719,-108.641,169.889,43.554,158.248
C03221=1033.123,201.471,-108.616,169.886,43.554,158.248
C03222=1033.117,201.223,-108.591,169.882,43.555,158.248
C03223=1033.111,200.974,-108.566,169.879,43.556,158.248
C03224=1033.104,200.725,-108.542,169.875,43.557,158.248
C03225=1033.099,200.476,-108.517,169.872,43.557,158.248
C03226=1033.093,200.228,-108.492,169.869,43.559,158.248
C03227=1033.086,199.979,-108.468,169.866,43.560,158.248
C03228=1033.080,199.730,-108.443,169.862,43.561,158.248
C03229=1033.074,199.481,-108.419,169.859,43.562,158.248
C03230=1033.068,199.233,-108.394,169.855,43.563,158.247
C03231=1033.061,198.984,-108.370,169.852,43.564,158.247
C03232=1033.055,198.735,-108.345,169.848,43.565,158.247
C03233=1033.048,198.487,-108.320,169.845,43.566,158.247
C03234=1033.043,198.238,-108.296,169.841,43.566,158.247
C03235=1033.036,197.989,-108.272,169.838,43.568,158.247
C03236=1033.030,197.740,-108.247,169.834,43.569,158.247
C03237=1033.024,197.492,-108.223,169.831,43.570,158.247
C03238=1033.018,197.243,-108.198,169.827,43.571,158.247
C03239=1033.012,196.994,-108.173,169.824,43.572,158.247
C03240=1033.005,196.745,-108.149,169.821,43.573,158.247
C03241=1033.000,196.497,-108.125,169.818,43.574,158.247
C03242=1032.993,196.248,-108.100,169.815,43.575,158.247
C03243=1032.987,195.999,-108.075,169.811,43.576,158.247
C03244=1032.981,195.751,-108.052,169.808,43.577,158.246
C03245=1032.975,195.501,-108.027,169.804,43.578,158.246
C03246=1032.968,195.253,-108.002,169.801,43.579,158.246
C03247=1032.963,195.005,-107.978,169.797,43.580,158.246
C03248=1032.957,194.756,-107.954,169.794,43.581,158.246
C03249=1032.951,194.506,-107.929,169.790,43.582,158.246
C03250=1032.944,194.259,-107.905,169.787,43.583,158.246
C03251=1032.938,194.009,-107.880,169.785,43.584,158.246
C03252=1032.932,193.761,-107.857,169.781,43.585,158.246
C03253=1032.926,193.512,-107.833,169.778,43.586,158.246
C03254=1032.920,193.263,-107.808,169.774,43.588,158.246
C03255=1032.914,193.015,-107.785,169.771,43.588,158.246
C03256=1032.908,192.766,-107.759,169.768,43.589,158.246
C03257=1032.902,192.518,-107.736,169.764,43.591,158.246
C03258=1032.896,192.268,-107.711,169.761,43.591,158.246
C03259=1032.890,192.020,-107.687,169.757,43.593,158.246
C03260=1032.884,191.771,-107.663,169.755,43.594,158.246
C03261=1032.877,191.522,-107.639,169.752,43.594,158.245
C03262=1032.872,191.273,-107.614,169.748,43.596,158.245
C03263=1032.865,191.024,-107.590,169.745,43.597,158.245
C03264=1032.860,190.776,-107.566,169.741,43.598,158.245
C03265=1032.853,190.527,-107.542,169.738,43.599,158.245
C03266=1032.848,190.278,-107.518,169.735,43.600,158.245
C03267=1032.841,190.029,-107.494,169.731,43.601,158.245
C03268=1032.836,189.780,-107.469,169.728,43.602,158.245
C03269=1032.829,189.531,-107.445,169.725,43.603,158.245
C03270=1032.824,189.283,-107.421,169.721,43.604,158.245
C03271=1032.817,189.000,-107.394,169.719,43.605,158.245
C03272=1032.810,188.716,-107.366,169.715,43.607,158.245
C03273=1032.803,188.431,-107.339,169.711,43.608,158.245
C03274=1032.796,188.148,-107.311,169.707,43.609,158.245
C03275=1032.791,187.899,-107.287,169.704,43.610,158.245
C03276=1032.784,187.650,-107.263,169.700,43.611,158.245
C03277=1032.779,187.402,-107.239,169.697,43.613,158.245
C03278=1032.772,187.153,-107.215,169.694,43.613,158.244
C03279=1032.766,186.904,-107.191,169.692,43.614,158.244
C03280=1032.761,186.656,-107.167,169.688,43.616,158.244
C03281=1032.754,186.406,-107.144,169.685,43.616,158.244
C03282=1032.749,186.158,-107.119,169.682,43.617,158.244
C03283=1032.742,185.909,-107.095,169.678,43.619,158.244
C03284=1032.737,185.660,-107.071,169.675,43.620,158.244
C03285=1032.731,185.412,-107.047,169.672,43.621,158.244
C03286=1032.725,185.162,-107.023,169.668,43.622,158.244
C03287=1032.719,184.914,-106.999,169.665,43.623,158.244
C03288=1032.713,184.665,-106.976,169.662,43.624,158.244
C03289=1032.708,184.416,-106.951,169.660,43.625,158.244
C03290=1032.702,184.168,-106.928,169.656,43.626,158.244
C03291=1032.696,183.919,-106.904,169.653,43.628,158.244
C03292=1032.690,183.670,-106.880,169.650,43.628,158.244
C03293=1032.685,183.421,-106.856,169.647,43.629,158.244
C03294=1032.679,183.173,-106.832,169.643,43.631,158.244
C03295=1032.672,182.924,-106.808,169.640,43.632,158.244
C03296=1032.666,182.675,-106.785,169.638,43.633,158.244
C03297=1032.660,182.426,-106.761,169.634,43.634,158.244
C03298=1032.654,182.177,-106.738,169.631,43.636,158.244
C03299=1032.646,181.928,-106.715,169.628,43.637,158.244
C03300=1032.641,181.679,-106.692,169.624,43.638,158.244
C03301=1032.635,181.431,-106.668,169.621,43.639,158.244
C03302=1032.628,181.182,-106.645,169.619,43.641,158.244
C03303=1032.622,180.933,-106.621,169.615,43.642,158.244
C03304=1032.616,180.684,-106.598,169.612,43.643,158.244
C03305=1032.610,180.435,-106.574,169.609,43.644,158.244
C03306=1032.603,180.187,-106.552,169.606,43.647,158.244
C03307=1032.597,179.938,-106.528,169.603,43.648,158.244
C03308=1032.591,179.689,-106.505,169.600,43.649,158.244
C03309=1032.585,179.440,-106.482,169.596,43.650,158.244
C03310=1032.579,179.191,-106.458,169.593,43.652,158.244
C03311=1032.573,178.942,-106.435,169.590,43.653,158.244
C03312=1032.566,178.693,-106.412,169.587,43.654,158.244
C03313=1032.560,178.445,-106.389,169.584,43.655,158.244
C03314=1032.554,178.196,-106.366,169.581,43.657,158.244
C03315=1032.548,177.947,-106.342,169.578,43.658,158.244
C03316=1032.542,177.698,-106.319,169.574,43.659,158.244
C03317=1032.536,177.449,-106.296,169.571,43.660,158.244
C03318=1032.529,177.201,-106.273,169.569,43.662,158.244
C03319=1032.523,176.951,-106.250,169.565,43.664,158.244
C03320=1032.517,176.702,-106.227,169.562,43.665,158.244
C03321=1032.511,176.454,-106.203,169.559,43.666,158.244
C03322=1032.505,176.205,-106.180,169.557,43.667,158.244
C03323=1032.499,175.956,-106.157,169.553,43.669,158.244
C03324=1032.492,175.708,-106.134,169.550,43.670,158.244
C03325=1032.487,175.459,-106.111,169.547,43.671,158.244
C03326=1032.480,175.209,-106.087,169.544,43.672,158.244
C03327=1032.475,174.960,-106.064,169.540,43.674,158.244
C03328=1032.469,174.712,-106.041,169.538,43.675,158.244
C03329=1032.462,174.463,-106.018,169.535,43.677,158.244
C03330=1032.456,174.214,-105.995,169.532,43.678,158.244
C03331=1032.450,173.965,-105.972,169.528,43.679,158.244
C03332=1032.444,173.716,-105.949,169.526,43.680,158.244
C03333=1032.438,173.468,-105.926,169.523,43.682,158.244
C03334=1032.432,173.219,-105.903,169.520,43.683,158.244
C03335=1032.426,172.934,-105.877,169.516,43.685,158.244
C03336=1032.418,172.651,-105.850,169.512,43.686,158.244
C03337=1032.411,172.366,-105.824,169.510,43.688,158.244
C03338=1032.404,172.081,-105.797,169.506,43.689,158.244
C03339=1032.398,171.833,-105.775,169.503,43.691,158.244
C03340=1032.392,171.584,-105.752,169.500,43.692,158.244
C03341=1032.386,171.336,-105.728,169.498,43.693,158.244
C03342=1032.381,171.087,-105.706,169.494,43.695,158.244
C03343=1032.374,170.838,-105.683,169.491,43.696,158.244
C03344=1032.368,170.589,-105.660,169.488,43.697,158.244
C03345=1032.362,170.340,-105.637,169.485,43.698,158.244
C03346=1032.356,170.091,-105.614,169.483,43.700,158.244
C03347=1032.351,169.842,-105.591,169.479,43.701,158.244
C03348=1032.344,169.593,-105.569,169.476,43.703,158.244
C03349=1032.338,169.344,-105.546,169.473,43.704,158.244
C03350=1032.333,169.095,-105.523,169.470,43.705,158.244
C03351=1032.327,168.847,-105.500,169.467,43.706,158.244
C03352=1032.321,168.598,-105.477,169.465,43.708,158.244
C03353=1032.315,168.349,-105.455,169.461,43.709,158.244
C03354=1032.308,168.099,-105.431,169.458,43.711,158.244
C03355=1032.303,167.851,-105.408,169.455,43.712,158.244
C03356=1032.297,167.602,-105.385,169.453,43.713,158.244
C03357=1032.290,167.353,-105.363,169.450,43.714,158.244
C03358=1032.285,167.104,-105.340,169.447,43.716,158.245
C03359=1032.279,166.855,-105.317,169.444,43.717,158.245
C03360=1032.273,166.606,-105.294,169.440,43.719,158.245
C03361=1032.267,166.358,-105.272,169.438,43.720,158.245
C03362=1032.261,166.109,-105.249,169.435,43.721,158.245
C03363=1032.255,165.860,-105.226,169.432,43.723,158.245
C03364=1032.250,165.611,-105.203,169.429,43.724,158.245
C03365=1032.243,165.362,-105.181,169.426,43.725,158.245
C03366=1032.237,165.114,-105.158,169.424,43.726,158.245
C03367=1032.232,164.864,-105.135,169.421,43.728,158.245
C03368=1032.226,164.615,-105.113,169.418,43.729,158.245
C03369=1032.220,164.366,-105.090,169.414,43.731,158.245
C03370=1032.214,164.118,-105.067,169.411,43.732,158.245
C03371=1032.208,163.869,-105.044,169.409,43.733,158.245
C03372=1032.203,163.620,-105.021,169.406,43.734,158.245
C03373=1032.197,163.371,-104.998,169.403,43.736,158.245
C03374=1032.191,163.122,-104.977,169.400,43.737,158.245
C03375=1032.185,162.873,-104.954,169.398,43.739,158.245
C03376=1032.179,162.624,-104.931,169.395,43.740,158.245
C03377=1032.173,162.375,-104.908,169.392,43.741,158.245
C03378=1032.167,162.127,-104.886,169.389,43.742,158.245
C03379=1032.162,161.877,-104.863,169.387,43.744,158.245
C03380=1032.156,161.628,-104.840,169.384,43.745,158.245
C03381=1032.150,161.380,-104.818,169.381,43.746,158.245
C03382=1032.144,161.131,-104.795,169.378,43.748,158.245
C03383=1032.139,160.882,-104.773,169.374,43.749,158.245
C03384=1032.133,160.633,-104.750,169.371,43.750,158.245
C03385=1032.127,160.384,-104.728,169.369,43.752,158.245
C03386=1032.121,160.135,-104.705,169.366,43.753,158.245
C03387=1032.115,159.886,-104.683,169.363,43.755,158.245
C03388=1032.110,159.637,-104.660,169.360,43.756,158.245
C03389=1032.104,159.388,-104.638,169.358,43.757,158.245
C03390=1032.097,159.139,-104.616,169.355,43.759,158.245
C03391=1032.091,158.891,-104.593,169.352,43.760,158.245
C03392=1032.085,158.641,-104.571,169.349,43.762,158.246
C03393=1032.079,158.393,-104.549,169.347,43.763,158.246
C03394=1032.073,158.143,-104.527,169.344,43.764,158.246
C03395=1032.067,157.895,-104.505,169.341,43.766,158.246
C03396=1032.061,157.646,-104.483,169.337,43.768,158.246
C03397=1032.055,157.397,-104.461,169.335,43.770,158.246
C03398=1032.049,157.148,-104.438,169.332,43.771,158.246
C03399=1032.042,156.864,-104.413,169.329,43.773,158.246
C03400=1032.035,156.579,-104.388,169.326,43.774,158.246
C03401=1032.028,156.294,-104.363,169.323,43.776,158.246
C03402=1032.022,156.009,-104.338,169.319,43.777,158.246
C03403=1032.015,155.761,-104.315,169.317,43.779,158.246
C03404=1032.010,155.511,-104.293,169.314,43.780,158.246
C03405=1032.003,155.262,-104.271,169.311,43.782,158.246
C03406=1031.997,155.013,-104.249,169.308,43.783,158.246
C03407=1031.991,154.764,-104.228,169.305,43.785,158.246
C03408=1031.986,154.516,-104.205,169.303,43.787,158.246
C03409=1031.980,154.267,-104.183,169.300,43.788,158.246
C03410=1031.973,154.018,-104.161,169.297,43.790,158.247
C03411=1031.968,153.768,-104.139,169.295,43.791,158.247
C03412=1031.962,153.519,-104.117,169.292,43.792,158.247
C03413=1031.955,153.271,-104.095,169.289,43.794,158.247
C03414=1031.949,153.021,-104.073,169.285,43.795,158.247
C03415=1031.943,152.773,-104.052,169.283,43.797,158.247
C03416=1031.937,152.524,-104.030,169.280,43.798,158.247
C03417=1031.931,152.275,-104.008,169.277,43.800,158.247
C03418=1031.925,152.026,-103.986,169.274,43.801,158.247
C03419=1031.919,151.776,-103.964,169.272,43.803,158.247
C03420=1031.913,151.527,-103.942,169.269,43.805,158.247
C03421=1031.907,151.279,-103.920,169.266,43.806,158.247
C03422=1031.901,151.030,-103.899,169.264,43.808,158.247
C03423=1031.895,150.781,-103.877,169.261,43.810,158.248
C03424=1031.889,150.532,-103.855,169.258,43.811,158.248
C03425=1031.883,150.283,-103.833,169.256,43.813,158.248
C03426=1031.877,150.034,-103.811,169.253,43.814,158.248
C03427=1031.871,149.785,-103.790,169.250,43.816,158.248
C03428=1031.865,149.536,-103.768,169.247,43.817,158.248
C03429=1031.859,149.287,-103.746,169.245,43.818,158.248
C03430=1031.853,149.038,-103.725,169.242,43.820,158.248
C03431=1031.847,148.790,-103.703,169.239,43.821,158.248
C03432=1031.841,148.540,-103.681,169.237,43.823,158.248
C03433=1031.835,148.291,-103.659,169.234,43.824,158.248
C03434=1031.829,148.042,-103.637,169.231,43.826,158.248
C03435=1031.824,147.793,-103.616,169.228,43.827,158.248
C03436=1031.817,147.544,-103.594,169.226,43.829,158.248
C03437=1031.811,147.295,-103.573,169.223,43.831,158.248
C03438=1031.805,147.046,-103.551,169.220,43.832,158.249
C03439=1031.800,146.797,-103.530,169.218,43.834,158.249
C03440=1031.793,146.548,-103.508,169.215,43.835,158.249
C03441=1031.787,146.299,-103.487,169.212,43.837,158.249
C03442=1031.781,146.049,-103.465,169.209,43.839,158.249
C03443=1031.775,145.801,-103.444,169.207,43.840,158.249
C03444=1031.769,145.552,-103.423,169.204,43.842,158.249
C03445=1031.762,145.303,-103.401,169.201,43.844,158.249
C03446=1031.756,145.054,-103.379,169.199,43.845,158.249
C03447=1031.751,144.805,-103.358,169.196,43.847,158.249
C03448=1031.745,144.556,-103.336,169.193,43.849,158.249
C03449=1031.738,144.307,-103.315,169.191,43.850,158.249
C03450=1031.733,144.058,-103.293,169.188,43.852,158.250
C03451=1031.727,143.809,-103.272,169.185,43.854,158.250
C03452=1031.720,143.560,-103.251,169.183,43.855,158.250
C03453=1031.714,143.312,-103.230,169.180,43.857,158.250
C03454=1031.708,143.062,-103.208,169.177,43.858,158.250
C03455=1031.702,142.813,-103.186,169.175,43.860,158.250
C03456=1031.696,142.563,-103.165,169.172,43.862,158.250
C03457=1031.690,142.315,-103.144,169.169,43.863,158.250
C03458=1031.684,142.066,-103.122,169.167,43.865,158.250
C03459=1031.677,141.817,-103.101,169.164,43.866,158.250
C03460=1031.672,141.568,-103.080,169.161,43.868,158.250
C03461=1031.666,141.319,-103.059,169.158,43.869,158.250
C03462=1031.660,141.071,-103.037,169.156,43.871,158.251
C03463=1031.653,140.785,-103.014,169.152,43.873,158.251
C03464=1031.647,140.500,-102.989,169.149,43.875,158.251
C03465=1031.639,140.215,-102.964,169.147,43.876,158.251
C03466=1031.633,139.930,-102.940,169.143,43.878,158.251
C03467=1031.626,139.681,-102.919,169.140,43.880,158.251
C03468=1031.620,139.432,-102.898,169.138,43.881,158.251
C03469=1031.614,139.183,-102.876,169.135,43.883,158.251
C03470=1031.609,138.934,-102.856,169.132,43.885,158.251
C03471=1031.603,138.685,-102.834,169.130,43.886,158.251
C03472=1031.596,138.436,-102.813,169.128,43.888,158.252
C03473=1031.590,138.187,-102.792,169.125,43.890,158.252
C03474=1031.585,137.938,-102.771,169.123,43.891,158.252
C03475=1031.578,137.689,-102.750,169.120,43.893,158.252
C03476=1031.572,137.440,-102.728,169.117,43.895,158.252
C03477=1031.566,137.190,-102.707,169.115,43.896,158.252
C03478=1031.561,136.942,-102.686,169.112,43.898,158.252
C03479=1031.554,136.693,-102.665,169.109,43.900,158.252
C03480=1031.549,136.444,-102.645,169.107,43.901,158.252
C03481=1031.542,136.195,-102.623,169.104,43.903,158.252
C03482=1031.536,135.945,-102.603,169.101,43.905,158.253
C03483=1031.530,135.697,-102.581,169.099,43.906,158.253
C03484=1031.523,135.448,-102.560,169.096,43.908,158.253
C03485=1031.518,135.199,-102.540,169.093,43.910,158.253
C03486=1031.512,134.949,-102.518,169.091,43.911,158.253
C03487=1031.506,134.701,-102.498,169.088,43.913,158.253
C03488=1031.500,134.451,-102.476,169.085,43.915,158.253
C03489=1031.493,134.202,-102.456,169.082,43.916,158.253
C03490=1031.488,133.953,-102.435,169.080,43.918,158.253
C03491=1031.482,133.703,-102.414,169.077,43.920,158.254
C03492=1031.475,133.455,-102.393,169.075,43.922,158.254
C03493=1031.470,133.205,-102.372,169.073,43.923,158.254
C03494=1031.463,132.957,-102.352,169.070,43.925,158.254
C03495=1031.457,132.707,-102.331,169.068,43.926,158.254
C03496=1031.452,132.459,-102.310,169.065,43.928,158.254
C03497=1031.445,132.209,-102.289,169.062,43.930,158.254
C03498=1031.440,131.961,-102.268,169.060,43.931,158.254
C03499=1031.433,131.711,-102.248,169.057,43.933,158.254
C03500=1031.428,131.463,-102.226,169.054,43.935,158.254
C03501=1031.421,131.213,-102.206,169.052,43.936,158.255
C03502=1031.415,130.965,-102.185,169.049,43.938,158.255
C03503=1031.410,130.715,-102.164,169.046,43.940,158.255
C03504=1031.404,130.466,-102.144,169.044,43.941,158.255
C03505=1031.397,130.217,-102.123,169.041,43.943,158.255
C03506=1031.391,129.968,-102.102,169.038,43.945,158.255
C03507=1031.385,129.719,-102.082,169.037,43.946,158.255
C03508=1031.378,129.471,-102.061,169.034,43.948,158.255
C03509=1031.372,129.221,-102.041,169.031,43.950,158.255
C03510=1031.366,128.971,-102.020,169.029,43.952,158.256
C03511=1031.360,128.723,-101.999,169.026,43.954,158.256
C03512=1031.353,128.473,-101.979,169.024,43.956,158.256
C03513=1031.347,128.225,-101.959,169.021,43.957,158.256
C03514=1031.342,127.976,-101.939,169.018,43.959,158.256
C03515=1031.335,127.727,-101.917,169.016,43.961,158.256
C03516=1031.329,127.478,-101.898,169.013,43.963,158.256
C03517=1031.323,127.228,-101.877,169.010,43.964,158.256
C03518=1031.317,126.979,-101.857,169.008,43.966,158.257
C03519=1031.311,126.730,-101.836,169.005,43.968,158.257
C03520=1031.304,126.481,-101.816,169.002,43.969,158.257
C03521=1031.298,126.232,-101.795,169.000,43.971,158.257
C03522=1031.292,125.983,-101.775,168.997,43.973,158.257
C03523=1031.286,125.733,-101.754,168.995,43.975,158.257
C03524=1031.280,125.484,-101.734,168.993,43.977,158.257
C03525=1031.274,125.235,-101.713,168.990,43.978,158.257
C03526=1031.268,124.986,-101.693,168.988,43.980,158.258
C03527=1031.261,124.701,-101.669,168.984,43.982,158.258
C03528=1031.253,124.417,-101.647,168.981,43.984,158.258
C03529=1031.247,124.131,-101.624,168.979,43.986,158.258
C03530=1031.240,123.845,-101.600,168.975,43.989,158.258
C03531=1031.233,123.597,-101.579,168.973,43.990,158.258
C03532=1031.227,123.348,-101.559,168.971,43.991,158.258
C03533=1031.221,123.099,-101.539,168.968,43.993,158.258
C03534=1031.216,122.850,-101.518,168.966,43.995,158.259
C03535=1031.209,122.600,-101.498,168.963,43.997,158.259
C03536=1031.203,122.351,-101.478,168.960,43.998,158.259
C03537=1031.197,122.103,-101.458,168.958,44.000,158.259
C03538=1031.191,121.853,-101.437,168.955,44.002,158.259
C03539=1031.185,121.604,-101.417,168.953,44.004,158.259
C03540=1031.179,121.355,-101.397,168.950,44.006,158.259
C03541=1031.173,121.106,-101.377,168.948,44.007,158.259
C03542=1031.167,120.856,-101.356,168.946,44.009,158.260
C03543=1031.161,120.608,-101.336,168.943,44.011,158.260
C03544=1031.155,120.358,-101.316,168.940,44.013,158.260
C03545=1031.149,120.109,-101.296,168.938,44.015,158.260
C03546=1031.143,119.860,-101.276,168.935,44.016,158.260
C03547=1031.137,119.611,-101.255,168.932,44.018,158.260
C03548=1031.131,119.362,-101.235,168.931,44.019,158.260
C03549=1031.125,119.113,-101.215,168.928,44.021,158.260
C03550=1031.118,118.864,-101.195,168.925,44.022,158.260
C03551=1031.113,118.614,-101.175,168.923,44.024,158.261
C03552=1031.107,118.366,-101.155,168.920,44.026,158.261
C03553=1031.100,118.116,-101.134,168.918,44.028,158.261
C03554=1031.094,117.867,-101.114,168.915,44.030,158.261
C03555=1031.088,117.618,-101.094,168.913,44.031,158.261
C03556=1031.083,117.369,-101.074,168.911,44.033,158.261
C03557=1031.077,117.120,-101.053,168.908,44.035,158.261
C03558=1031.071,116.871,-101.033,168.905,44.037,158.261
C03559=1031.065,116.622,-101.014,168.903,44.038,158.261
C03560=1031.058,116.373,-100.993,168.900,44.040,158.262
C03561=1031.053,116.124,-100.973,168.899,44.042,158.262
C03562=1031.047,115.875,-100.953,168.896,44.044,158.262
C03563=1031.041,115.626,-100.933,168.893,44.045,158.262
C03564=1031.035,115.376,-100.913,168.890,44.047,158.262
C03565=1031.029,115.127,-100.893,168.888,44.049,158.262
C03566=1031.023,114.878,-100.873,168.885,44.050,158.262
C03567=1031.017,114.629,-100.853,168.883,44.052,158.262
C03568=1031.011,114.380,-100.833,168.881,44.053,158.262
C03569=1031.005,114.131,-100.812,168.878,44.055,158.263
C03570=1030.999,113.882,-100.792,168.876,44.057,158.263
C03571=1030.994,113.632,-100.773,168.873,44.058,158.263
C03572=1030.988,113.383,-100.753,168.871,44.060,158.263
C03573=1030.981,113.134,-100.732,168.869,44.062,158.263
C03574=1030.975,112.885,-100.712,168.866,44.064,158.263
C03575=1030.969,112.636,-100.693,168.864,44.066,158.263
C03576=1030.963,112.387,-100.673,168.861,44.067,158.263
C03577=1030.957,112.137,-100.653,168.858,44.069,158.264
C03578=1030.951,111.888,-100.634,168.857,44.071,158.264
C03579=1030.945,111.639,-100.614,168.854,44.073,158.264
C03580=1030.939,111.390,-100.594,168.851,44.074,158.264
C03581=1030.934,111.141,-100.574,168.849,44.076,158.264
C03582=1030.927,110.891,-100.554,168.846,44.078,158.264
C03583=1030.921,110.642,-100.534,168.844,44.080,158.264
